// Communication
	fbReadWriteReq(sNetID := sNetID, nPort := nPort, nIdxGroup := nIdxGroup, tTimeOut := tTimeOut, aData := aStatIOLRecords);
	bStatTriggerExecute := bExecute AND NOT bStatTriggerExecuteMem;
	bStatTriggerExecuteMem := bExecute;
	bStatTriggerError := fbReadWriteReq.bError AND NOT bStatTriggerErrorMem;
	bStatTriggerErrorMem := fbReadWriteReq.bError;
// Timer
	fbInstTimeOut(IN:= bStatBusyMem, PT := tTimeOut);
// Error management
	IF stStatLastErrorCode.nBlockError <> cDEFAULT OR stStatLastErrorCode.nAdsReadError <> cDEFAULT OR stStatLastErrorCode.nAdsWriteError <> cDEFAULT THEN
		bDone := FALSE;
		bBusy := FALSE;
		bStatBusyMem := FALSE;
		bError := TRUE;
		stErrorCode := stStatLastErrorCode;
		stStatLastErrorCode.nBlockError := cDEFAULT;
		stStatLastErrorCode.nAdsReadError := cDEFAULT;
		stStatLastErrorCode.nAdsWriteError := cDEFAULT;
		stStatLastErrorCode.nIndex := 0;
		stStatLastErrorCode.nSubIndex := 0;
		nStatState := cSTATE_READY;
		RETURN;
	END_IF;
	IF bStatTriggerError THEN
		stStatLastErrorCode := fbReadWriteReq.stErrorCode;          // Error: ADS error
		RETURN;
	END_IF
	IF fbInstTimeOut.Q THEN
		stStatLastErrorCode.nIndex := fbReadWriteReq.stErrorCode.nIndex;
		stStatLastErrorCode.nSubIndex := fbReadWriteReq.stErrorCode.nSubIndex;
		stStatLastErrorCode.nBlockError := cERR_TIME_OUT;			// Error: Time out detected  
		RETURN;
	END_IF;
// Start R/W request
	IF bStatTriggerExecute AND NOT bStatBusyMem THEN
		bStatSource := FALSE; 
		nStatBitLength := 0; 
		nStatIndex := 0; 
		bDone := FALSE; 
		bBusy := TRUE; 
		bStatBusyMem := TRUE; 
		bError := FALSE; 
		stErrorCode.nBlockError := cDEFAULT; 
		stErrorCode.nAdsReadError := cDEFAULT; 
		stErrorCode.nAdsWriteError := cDEFAULT; 
		stErrorCode.nIndex := 0; 
		stErrorCode.nSubIndex := 0; 
		stStatLastErrorCode.nBlockError := cDEFAULT; 
		stStatLastErrorCode.nAdsReadError := cDEFAULT; 
		stStatLastErrorCode.nAdsWriteError := cDEFAULT; 
		stStatLastErrorCode.nIndex := 0; 
		stStatLastErrorCode.nSubIndex := 0; 
		bStatRWSave := bRW;
		nStatCommandIndex := 0;
		// Store input selection flags internally 
		aStatInputSelections[0] := stDeviceData.stSelection.stCommands.bCmdRestoreFactorySettings;
		aStatInputSelections[1] := stDeviceData.stSelection.stCommands.bCmdTeachApply;
		aStatInputSelections[2] := stDeviceData.stSelection.stCommands.bCmdSetpoint1SingleValueTeach;
		aStatInputSelections[3] := stDeviceData.stSelection.stCommands.bCmdSetpoint2SingleValueTeach;
		aStatInputSelections[4] := stDeviceData.stSelection.stCommands.bCmdTwoValueTeachTp1Sp1;
		aStatInputSelections[5] := stDeviceData.stSelection.stCommands.bCmdTwoValueTeachTp2Sp1;
		aStatInputSelections[6] := stDeviceData.stSelection.stCommands.bCmdTwoValueTeachTp1Sp2;
		aStatInputSelections[7] := stDeviceData.stSelection.stCommands.bCmdTwoValueTeachTp2Sp2;
		aStatInputSelections[8] := stDeviceData.stSelection.stCommands.bCmdSetpoint1DynamicTeachStart;
		aStatInputSelections[9] := stDeviceData.stSelection.stCommands.bCmdSetpoint1DynamicTeachStop;
		aStatInputSelections[10] := stDeviceData.stSelection.stCommands.bCmdSetpoint2DynamicTeachStart;
		aStatInputSelections[11] := stDeviceData.stSelection.stCommands.bCmdSetpoint2DynamicTeachStop;
		aStatInputSelections[12] := stDeviceData.stSelection.stCommands.bCmdTeachCancel;
		aStatInputSelections[13] := stDeviceData.stSelection.stCommands.bCmdSetAnalogOutputLowerLimit;
		aStatInputSelections[14] := stDeviceData.stSelection.stCommands.bCmdSetAnalogOutputUpperLimit;
		aStatInputSelections[15] := stDeviceData.stSelection.stCommands.bCmdResetDiagnosisInformation;
		aStatInputSelections[16] := stDeviceData.stSelection.stCommands.bCmdStopMeasurement;
		aStatInputSelections[17] := stDeviceData.stSelection.stCommands.bCmdStartMeasurement;
		aStatInputSelections[18] := stDeviceData.stSelection.stCommands.bCmdSingleMeasurement;
		aStatInputSelections[19] := stDeviceData.stSelection.stCommands.bCmdIoLink11SystemTestCommand240Event8DfeAppears;
		aStatInputSelections[20] := stDeviceData.stSelection.stCommands.bCmdIoLink11SystemTestCommand241Event8DfeDisappears;
		aStatInputSelections[21] := stDeviceData.stSelection.stCommands.bCmdIoLink11SystemTestCommand242Event8DffAppears;
		aStatInputSelections[22] := stDeviceData.stSelection.stCommands.bCmdIoLink11SystemTestCommand243Event8DffDisappears;
		aStatInputSelections[23] := stDeviceData.stSelection.stDirectParametersPage1.bAll;
		aStatInputSelections[24] := stDeviceData.stSelection.stDirectParametersPage1.bReserved_1;
		aStatInputSelections[25] := stDeviceData.stSelection.stDirectParametersPage1.bMasterCycleTime;
		aStatInputSelections[26] := stDeviceData.stSelection.stDirectParametersPage1.bMinCycleTime;
		aStatInputSelections[27] := stDeviceData.stSelection.stDirectParametersPage1.bMSequenceCapability;
		aStatInputSelections[28] := stDeviceData.stSelection.stDirectParametersPage1.bIoLinkRevisionId;
		aStatInputSelections[29] := stDeviceData.stSelection.stDirectParametersPage1.bProcessDataInputLength;
		aStatInputSelections[30] := stDeviceData.stSelection.stDirectParametersPage1.bProcessDataOutputLength;
		aStatInputSelections[31] := stDeviceData.stSelection.stDirectParametersPage1.bVendorId1;
		aStatInputSelections[32] := stDeviceData.stSelection.stDirectParametersPage1.bVendorId2;
		aStatInputSelections[33] := stDeviceData.stSelection.stDirectParametersPage1.bDeviceId1;
		aStatInputSelections[34] := stDeviceData.stSelection.stDirectParametersPage1.bDeviceId2;
		aStatInputSelections[35] := stDeviceData.stSelection.stDirectParametersPage1.bDeviceId3;
		aStatInputSelections[36] := stDeviceData.stSelection.stDirectParametersPage1.bReserved_13;
		aStatInputSelections[37] := stDeviceData.stSelection.stDirectParametersPage1.bReserved_14;
		aStatInputSelections[38] := stDeviceData.stSelection.stDirectParametersPage1.bReserved_15;
		aStatInputSelections[39] := stDeviceData.stSelection.stDirectParametersPage1.bSystemCommand;
		aStatInputSelections[40] := stDeviceData.stSelection.stDirectParametersPage2.bAll;
		aStatInputSelections[41] := stDeviceData.stSelection.stDirectParametersPage2.bDeviceSpecificParameter1;
		aStatInputSelections[42] := stDeviceData.stSelection.stDirectParametersPage2.bDeviceSpecificParameter2;
		aStatInputSelections[43] := stDeviceData.stSelection.stDirectParametersPage2.bDeviceSpecificParameter3;
		aStatInputSelections[44] := stDeviceData.stSelection.stDirectParametersPage2.bDeviceSpecificParameter4;
		aStatInputSelections[45] := stDeviceData.stSelection.stDirectParametersPage2.bDeviceSpecificParameter5;
		aStatInputSelections[46] := stDeviceData.stSelection.stDirectParametersPage2.bDeviceSpecificParameter6;
		aStatInputSelections[47] := stDeviceData.stSelection.stDirectParametersPage2.bDeviceSpecificParameter7;
		aStatInputSelections[48] := stDeviceData.stSelection.stDirectParametersPage2.bDeviceSpecificParameter8;
		aStatInputSelections[49] := stDeviceData.stSelection.stDirectParametersPage2.bDeviceSpecificParameter9;
		aStatInputSelections[50] := stDeviceData.stSelection.stDirectParametersPage2.bDeviceSpecificParameter10;
		aStatInputSelections[51] := stDeviceData.stSelection.stDirectParametersPage2.bDeviceSpecificParameter11;
		aStatInputSelections[52] := stDeviceData.stSelection.stDirectParametersPage2.bDeviceSpecificParameter12;
		aStatInputSelections[53] := stDeviceData.stSelection.stDirectParametersPage2.bDeviceSpecificParameter13;
		aStatInputSelections[54] := stDeviceData.stSelection.stDirectParametersPage2.bDeviceSpecificParameter14;
		aStatInputSelections[55] := stDeviceData.stSelection.stDirectParametersPage2.bDeviceSpecificParameter15;
		aStatInputSelections[56] := stDeviceData.stSelection.stDirectParametersPage2.bDeviceSpecificParameter16;
		aStatInputSelections[57] := stDeviceData.stSelection.bSystemCommand;
		aStatInputSelections[58] := stDeviceData.stSelection.stDeviceAccessLocks.bAll;
		aStatInputSelections[59] := stDeviceData.stSelection.bVendorName;
		aStatInputSelections[60] := stDeviceData.stSelection.bVendorText;
		aStatInputSelections[61] := stDeviceData.stSelection.bProductName;
		aStatInputSelections[62] := stDeviceData.stSelection.bProductId;
		aStatInputSelections[63] := stDeviceData.stSelection.bProductText;
		aStatInputSelections[64] := stDeviceData.stSelection.bFirmwareRevision;
		aStatInputSelections[65] := stDeviceData.stSelection.bApplicationSpecificTag;
		aStatInputSelections[66] := stDeviceData.stSelection.bErrorCount;
		aStatInputSelections[67] := stDeviceData.stSelection.bDeviceStatus;
		aStatInputSelections[68] := stDeviceData.stSelection.bTeachInSelect;
		aStatInputSelections[69] := stDeviceData.stSelection.stTeachState.bAll;
		aStatInputSelections[70] := stDeviceData.stSelection.stSetpoints_60.bAll;
		aStatInputSelections[71] := stDeviceData.stSelection.stSetpoints_60.bParam1Bdc1Q1;
		aStatInputSelections[72] := stDeviceData.stSelection.stSetpoints_60.bParam2Bdc1Q1;
		aStatInputSelections[73] := stDeviceData.stSelection.stSwitchpointBdc1.bAll;
		aStatInputSelections[74] := stDeviceData.stSelection.stSwitchpointBdc1.bLogic;
		aStatInputSelections[75] := stDeviceData.stSelection.stSwitchpointBdc1.bMode;
		aStatInputSelections[76] := stDeviceData.stSelection.stSwitchpointBdc1.bHysteresis;
		aStatInputSelections[77] := stDeviceData.stSelection.stSetpoints_62.bAll;
		aStatInputSelections[78] := stDeviceData.stSelection.stSetpoints_62.bParam1Bdc2Q2;
		aStatInputSelections[79] := stDeviceData.stSelection.stSetpoints_62.bParam2Bdc2Q2;
		aStatInputSelections[80] := stDeviceData.stSelection.stSwitchpointBdc2.bAll;
		aStatInputSelections[81] := stDeviceData.stSelection.stSwitchpointBdc2.bLogic;
		aStatInputSelections[82] := stDeviceData.stSelection.stSwitchpointBdc2.bMode;
		aStatInputSelections[83] := stDeviceData.stSelection.stSwitchpointBdc2.bHysteresis;
		aStatInputSelections[84] := stDeviceData.stSelection.bLot;
		aStatInputSelections[85] := stDeviceData.stSelection.bOnDelaySwitchingOutput;
		aStatInputSelections[86] := stDeviceData.stSelection.bOffDelaySwitchingOutput;
		aStatInputSelections[87] := stDeviceData.stSelection.bMultiIOPin4;
		aStatInputSelections[88] := stDeviceData.stSelection.bMultiIOPin2;
		aStatInputSelections[89] := stDeviceData.stSelection.stAnalogRange.bAll;
		aStatInputSelections[90] := stDeviceData.stSelection.stAnalogRange.bLowerLimit;
		aStatInputSelections[91] := stDeviceData.stSelection.stAnalogRange.bUpperLimit;
		aStatInputSelections[92] := stDeviceData.stSelection.bTemperatureCompensation;
		aStatInputSelections[93] := stDeviceData.stSelection.stTeachpointSp1_80.bAll;
		aStatInputSelections[94] := stDeviceData.stSelection.stTeachpointSp1_80.bTp1;
		aStatInputSelections[95] := stDeviceData.stSelection.stTeachpointSp1_80.bTp2;
		aStatInputSelections[96] := stDeviceData.stSelection.stTeachpointSp2_81.bAll;
		aStatInputSelections[97] := stDeviceData.stSelection.stTeachpointSp2_81.bTp1;
		aStatInputSelections[98] := stDeviceData.stSelection.stTeachpointSp2_81.bTp2;
		aStatInputSelections[99] := stDeviceData.stSelection.stTeachpointSp1_82.bAll;
		aStatInputSelections[100] := stDeviceData.stSelection.stTeachpointSp1_82.bTp1;
		aStatInputSelections[101] := stDeviceData.stSelection.stTeachpointSp1_82.bTp2;
		aStatInputSelections[102] := stDeviceData.stSelection.stTeachpointSp2_83.bAll;
		aStatInputSelections[103] := stDeviceData.stSelection.stTeachpointSp2_83.bTp1;
		aStatInputSelections[104] := stDeviceData.stSelection.stTeachpointSp2_83.bTp2;
		aStatInputSelections[105] := stDeviceData.stSelection.stProcessDataLimits.bAll;
		aStatInputSelections[106] := stDeviceData.stSelection.stProcessDataLimits.bLower;
		aStatInputSelections[107] := stDeviceData.stSelection.stProcessDataLimits.bUpper;
		aStatInputSelections[108] := stDeviceData.stSelection.bSwitchCounter;
		aStatInputSelections[109] := stDeviceData.stSelection.bTemperatureInternal;
		aStatInputSelections[110] := stDeviceData.stSelection.stNetwork.bAll;
		aStatInputSelections[111] := stDeviceData.stSelection.stNetwork.bRoleInNetwork;
		aStatInputSelections[112] := stDeviceData.stSelection.stNetwork.bDeviceNoMasterHighestNo;
		nStatState := cSTATE_INIT;
		RETURN; // Show the Busy-Flag for at least one PLC cycle 
	END_IF;
// Create command queue
	IF nStatState = cSTATE_INIT THEN
		// Check number of selected input selection bits
		nStatNumSelection := 0;
		FOR nTempLoopIndex := 0 TO cNUMBER_INPUTS DO
			IF aStatInputSelections[nTempLoopIndex] THEN
				nStatNumSelection := nStatNumSelection + 1;
			END_IF;
		END_FOR;
		IF nStatNumSelection = 0 THEN
			stStatLastErrorCode.nBlockError := cERR_EMPTY_SELECTION;
			RETURN;
		END_IF;
		// Create command queue
		FOR nTempLoopIndex := 0 TO cNUMBER_INPUTS DO
			aStatCommandQueue[nTempLoopIndex].nIndex := cEMPTY_COMMAND_QUEUE;
		END_FOR;
		nTempLoopIndex := 0;
		// stCommands - bCmdRestoreFactorySettings [BOOL] [WRITE_ONLY]
		IF aStatInputSelections[0] THEN
			aStatCommandQueue[nTempLoopIndex].nIndex := 32767;
			aStatCommandQueue[nTempLoopIndex].nSubIndex := 1;
			aStatCommandQueue[nTempLoopIndex].nBitLength := 8;
			nTempLoopIndex := nTempLoopIndex + 1;
		END_IF;
		// stCommands - bCmdTeachApply [BOOL] [WRITE_ONLY]
		IF aStatInputSelections[1] THEN
			aStatCommandQueue[nTempLoopIndex].nIndex := 32767;
			aStatCommandQueue[nTempLoopIndex].nSubIndex := 2;
			aStatCommandQueue[nTempLoopIndex].nBitLength := 8;
			nTempLoopIndex := nTempLoopIndex + 1;
		END_IF;
		// stCommands - bCmdSetpoint1SingleValueTeach [BOOL] [WRITE_ONLY]
		IF aStatInputSelections[2] THEN
			aStatCommandQueue[nTempLoopIndex].nIndex := 32767;
			aStatCommandQueue[nTempLoopIndex].nSubIndex := 3;
			aStatCommandQueue[nTempLoopIndex].nBitLength := 8;
			nTempLoopIndex := nTempLoopIndex + 1;
		END_IF;
		// stCommands - bCmdSetpoint2SingleValueTeach [BOOL] [WRITE_ONLY]
		IF aStatInputSelections[3] THEN
			aStatCommandQueue[nTempLoopIndex].nIndex := 32767;
			aStatCommandQueue[nTempLoopIndex].nSubIndex := 4;
			aStatCommandQueue[nTempLoopIndex].nBitLength := 8;
			nTempLoopIndex := nTempLoopIndex + 1;
		END_IF;
		// stCommands - bCmdTwoValueTeachTp1Sp1 [BOOL] [WRITE_ONLY]
		IF aStatInputSelections[4] THEN
			aStatCommandQueue[nTempLoopIndex].nIndex := 32767;
			aStatCommandQueue[nTempLoopIndex].nSubIndex := 5;
			aStatCommandQueue[nTempLoopIndex].nBitLength := 8;
			nTempLoopIndex := nTempLoopIndex + 1;
		END_IF;
		// stCommands - bCmdTwoValueTeachTp2Sp1 [BOOL] [WRITE_ONLY]
		IF aStatInputSelections[5] THEN
			aStatCommandQueue[nTempLoopIndex].nIndex := 32767;
			aStatCommandQueue[nTempLoopIndex].nSubIndex := 6;
			aStatCommandQueue[nTempLoopIndex].nBitLength := 8;
			nTempLoopIndex := nTempLoopIndex + 1;
		END_IF;
		// stCommands - bCmdTwoValueTeachTp1Sp2 [BOOL] [WRITE_ONLY]
		IF aStatInputSelections[6] THEN
			aStatCommandQueue[nTempLoopIndex].nIndex := 32767;
			aStatCommandQueue[nTempLoopIndex].nSubIndex := 7;
			aStatCommandQueue[nTempLoopIndex].nBitLength := 8;
			nTempLoopIndex := nTempLoopIndex + 1;
		END_IF;
		// stCommands - bCmdTwoValueTeachTp2Sp2 [BOOL] [WRITE_ONLY]
		IF aStatInputSelections[7] THEN
			aStatCommandQueue[nTempLoopIndex].nIndex := 32767;
			aStatCommandQueue[nTempLoopIndex].nSubIndex := 8;
			aStatCommandQueue[nTempLoopIndex].nBitLength := 8;
			nTempLoopIndex := nTempLoopIndex + 1;
		END_IF;
		// stCommands - bCmdSetpoint1DynamicTeachStart [BOOL] [WRITE_ONLY]
		IF aStatInputSelections[8] THEN
			aStatCommandQueue[nTempLoopIndex].nIndex := 32767;
			aStatCommandQueue[nTempLoopIndex].nSubIndex := 9;
			aStatCommandQueue[nTempLoopIndex].nBitLength := 8;
			nTempLoopIndex := nTempLoopIndex + 1;
		END_IF;
		// stCommands - bCmdSetpoint1DynamicTeachStop [BOOL] [WRITE_ONLY]
		IF aStatInputSelections[9] THEN
			aStatCommandQueue[nTempLoopIndex].nIndex := 32767;
			aStatCommandQueue[nTempLoopIndex].nSubIndex := 10;
			aStatCommandQueue[nTempLoopIndex].nBitLength := 8;
			nTempLoopIndex := nTempLoopIndex + 1;
		END_IF;
		// stCommands - bCmdSetpoint2DynamicTeachStart [BOOL] [WRITE_ONLY]
		IF aStatInputSelections[10] THEN
			aStatCommandQueue[nTempLoopIndex].nIndex := 32767;
			aStatCommandQueue[nTempLoopIndex].nSubIndex := 11;
			aStatCommandQueue[nTempLoopIndex].nBitLength := 8;
			nTempLoopIndex := nTempLoopIndex + 1;
		END_IF;
		// stCommands - bCmdSetpoint2DynamicTeachStop [BOOL] [WRITE_ONLY]
		IF aStatInputSelections[11] THEN
			aStatCommandQueue[nTempLoopIndex].nIndex := 32767;
			aStatCommandQueue[nTempLoopIndex].nSubIndex := 12;
			aStatCommandQueue[nTempLoopIndex].nBitLength := 8;
			nTempLoopIndex := nTempLoopIndex + 1;
		END_IF;
		// stCommands - bCmdTeachCancel [BOOL] [WRITE_ONLY]
		IF aStatInputSelections[12] THEN
			aStatCommandQueue[nTempLoopIndex].nIndex := 32767;
			aStatCommandQueue[nTempLoopIndex].nSubIndex := 13;
			aStatCommandQueue[nTempLoopIndex].nBitLength := 8;
			nTempLoopIndex := nTempLoopIndex + 1;
		END_IF;
		// stCommands - bCmdSetAnalogOutputLowerLimit [BOOL] [WRITE_ONLY]
		IF aStatInputSelections[13] THEN
			aStatCommandQueue[nTempLoopIndex].nIndex := 32767;
			aStatCommandQueue[nTempLoopIndex].nSubIndex := 14;
			aStatCommandQueue[nTempLoopIndex].nBitLength := 8;
			nTempLoopIndex := nTempLoopIndex + 1;
		END_IF;
		// stCommands - bCmdSetAnalogOutputUpperLimit [BOOL] [WRITE_ONLY]
		IF aStatInputSelections[14] THEN
			aStatCommandQueue[nTempLoopIndex].nIndex := 32767;
			aStatCommandQueue[nTempLoopIndex].nSubIndex := 15;
			aStatCommandQueue[nTempLoopIndex].nBitLength := 8;
			nTempLoopIndex := nTempLoopIndex + 1;
		END_IF;
		// stCommands - bCmdResetDiagnosisInformation [BOOL] [WRITE_ONLY]
		IF aStatInputSelections[15] THEN
			aStatCommandQueue[nTempLoopIndex].nIndex := 32767;
			aStatCommandQueue[nTempLoopIndex].nSubIndex := 16;
			aStatCommandQueue[nTempLoopIndex].nBitLength := 8;
			nTempLoopIndex := nTempLoopIndex + 1;
		END_IF;
		// stCommands - bCmdStopMeasurement [BOOL] [WRITE_ONLY]
		IF aStatInputSelections[16] THEN
			aStatCommandQueue[nTempLoopIndex].nIndex := 32767;
			aStatCommandQueue[nTempLoopIndex].nSubIndex := 17;
			aStatCommandQueue[nTempLoopIndex].nBitLength := 8;
			nTempLoopIndex := nTempLoopIndex + 1;
		END_IF;
		// stCommands - bCmdStartMeasurement [BOOL] [WRITE_ONLY]
		IF aStatInputSelections[17] THEN
			aStatCommandQueue[nTempLoopIndex].nIndex := 32767;
			aStatCommandQueue[nTempLoopIndex].nSubIndex := 18;
			aStatCommandQueue[nTempLoopIndex].nBitLength := 8;
			nTempLoopIndex := nTempLoopIndex + 1;
		END_IF;
		// stCommands - bCmdSingleMeasurement [BOOL] [WRITE_ONLY]
		IF aStatInputSelections[18] THEN
			aStatCommandQueue[nTempLoopIndex].nIndex := 32767;
			aStatCommandQueue[nTempLoopIndex].nSubIndex := 19;
			aStatCommandQueue[nTempLoopIndex].nBitLength := 8;
			nTempLoopIndex := nTempLoopIndex + 1;
		END_IF;
		// stCommands - bCmdIoLink11SystemTestCommand240Event8DfeAppears [BOOL] [WRITE_ONLY]
		IF aStatInputSelections[19] THEN
			aStatCommandQueue[nTempLoopIndex].nIndex := 32767;
			aStatCommandQueue[nTempLoopIndex].nSubIndex := 20;
			aStatCommandQueue[nTempLoopIndex].nBitLength := 8;
			nTempLoopIndex := nTempLoopIndex + 1;
		END_IF;
		// stCommands - bCmdIoLink11SystemTestCommand241Event8DfeDisappears [BOOL] [WRITE_ONLY]
		IF aStatInputSelections[20] THEN
			aStatCommandQueue[nTempLoopIndex].nIndex := 32767;
			aStatCommandQueue[nTempLoopIndex].nSubIndex := 21;
			aStatCommandQueue[nTempLoopIndex].nBitLength := 8;
			nTempLoopIndex := nTempLoopIndex + 1;
		END_IF;
		// stCommands - bCmdIoLink11SystemTestCommand242Event8DffAppears [BOOL] [WRITE_ONLY]
		IF aStatInputSelections[21] THEN
			aStatCommandQueue[nTempLoopIndex].nIndex := 32767;
			aStatCommandQueue[nTempLoopIndex].nSubIndex := 22;
			aStatCommandQueue[nTempLoopIndex].nBitLength := 8;
			nTempLoopIndex := nTempLoopIndex + 1;
		END_IF;
		// stCommands - bCmdIoLink11SystemTestCommand243Event8DffDisappears [BOOL] [WRITE_ONLY]
		IF aStatInputSelections[22] THEN
			aStatCommandQueue[nTempLoopIndex].nIndex := 32767;
			aStatCommandQueue[nTempLoopIndex].nSubIndex := 23;
			aStatCommandQueue[nTempLoopIndex].nBitLength := 8;
			nTempLoopIndex := nTempLoopIndex + 1;
		END_IF;
		// stDirectParametersPage1 - bAll [BOOL] [READ_WRITE]
		IF aStatInputSelections[23] THEN
			aStatCommandQueue[nTempLoopIndex].nIndex := 0;
			aStatCommandQueue[nTempLoopIndex].nSubIndex := 0;
			aStatCommandQueue[nTempLoopIndex].nBitLength := 128;
			nTempLoopIndex := nTempLoopIndex + 1;
		END_IF;
		// stDirectParametersPage1 - bReserved_1 [BOOL] [READ_ONLY]
		IF aStatInputSelections[24] THEN
			aStatCommandQueue[nTempLoopIndex].nIndex := 0;
			aStatCommandQueue[nTempLoopIndex].nSubIndex := 1;
			aStatCommandQueue[nTempLoopIndex].nBitLength := 8;
			nTempLoopIndex := nTempLoopIndex + 1;
		END_IF;
		// stDirectParametersPage1 - bMasterCycleTime [BOOL] [READ_ONLY]
		IF aStatInputSelections[25] THEN
			aStatCommandQueue[nTempLoopIndex].nIndex := 0;
			aStatCommandQueue[nTempLoopIndex].nSubIndex := 2;
			aStatCommandQueue[nTempLoopIndex].nBitLength := 8;
			nTempLoopIndex := nTempLoopIndex + 1;
		END_IF;
		// stDirectParametersPage1 - bMinCycleTime [BOOL] [READ_ONLY]
		IF aStatInputSelections[26] THEN
			aStatCommandQueue[nTempLoopIndex].nIndex := 0;
			aStatCommandQueue[nTempLoopIndex].nSubIndex := 3;
			aStatCommandQueue[nTempLoopIndex].nBitLength := 8;
			nTempLoopIndex := nTempLoopIndex + 1;
		END_IF;
		// stDirectParametersPage1 - bMSequenceCapability [BOOL] [READ_ONLY]
		IF aStatInputSelections[27] THEN
			aStatCommandQueue[nTempLoopIndex].nIndex := 0;
			aStatCommandQueue[nTempLoopIndex].nSubIndex := 4;
			aStatCommandQueue[nTempLoopIndex].nBitLength := 8;
			nTempLoopIndex := nTempLoopIndex + 1;
		END_IF;
		// stDirectParametersPage1 - bIoLinkRevisionId [BOOL] [READ_ONLY]
		IF aStatInputSelections[28] THEN
			aStatCommandQueue[nTempLoopIndex].nIndex := 0;
			aStatCommandQueue[nTempLoopIndex].nSubIndex := 5;
			aStatCommandQueue[nTempLoopIndex].nBitLength := 8;
			nTempLoopIndex := nTempLoopIndex + 1;
		END_IF;
		// stDirectParametersPage1 - bProcessDataInputLength [BOOL] [READ_ONLY]
		IF aStatInputSelections[29] THEN
			aStatCommandQueue[nTempLoopIndex].nIndex := 0;
			aStatCommandQueue[nTempLoopIndex].nSubIndex := 6;
			aStatCommandQueue[nTempLoopIndex].nBitLength := 8;
			nTempLoopIndex := nTempLoopIndex + 1;
		END_IF;
		// stDirectParametersPage1 - bProcessDataOutputLength [BOOL] [READ_ONLY]
		IF aStatInputSelections[30] THEN
			aStatCommandQueue[nTempLoopIndex].nIndex := 0;
			aStatCommandQueue[nTempLoopIndex].nSubIndex := 7;
			aStatCommandQueue[nTempLoopIndex].nBitLength := 8;
			nTempLoopIndex := nTempLoopIndex + 1;
		END_IF;
		// stDirectParametersPage1 - bVendorId1 [BOOL] [READ_ONLY]
		IF aStatInputSelections[31] THEN
			aStatCommandQueue[nTempLoopIndex].nIndex := 0;
			aStatCommandQueue[nTempLoopIndex].nSubIndex := 8;
			aStatCommandQueue[nTempLoopIndex].nBitLength := 8;
			nTempLoopIndex := nTempLoopIndex + 1;
		END_IF;
		// stDirectParametersPage1 - bVendorId2 [BOOL] [READ_ONLY]
		IF aStatInputSelections[32] THEN
			aStatCommandQueue[nTempLoopIndex].nIndex := 0;
			aStatCommandQueue[nTempLoopIndex].nSubIndex := 9;
			aStatCommandQueue[nTempLoopIndex].nBitLength := 8;
			nTempLoopIndex := nTempLoopIndex + 1;
		END_IF;
		// stDirectParametersPage1 - bDeviceId1 [BOOL] [READ_ONLY]
		IF aStatInputSelections[33] THEN
			aStatCommandQueue[nTempLoopIndex].nIndex := 0;
			aStatCommandQueue[nTempLoopIndex].nSubIndex := 10;
			aStatCommandQueue[nTempLoopIndex].nBitLength := 8;
			nTempLoopIndex := nTempLoopIndex + 1;
		END_IF;
		// stDirectParametersPage1 - bDeviceId2 [BOOL] [READ_ONLY]
		IF aStatInputSelections[34] THEN
			aStatCommandQueue[nTempLoopIndex].nIndex := 0;
			aStatCommandQueue[nTempLoopIndex].nSubIndex := 11;
			aStatCommandQueue[nTempLoopIndex].nBitLength := 8;
			nTempLoopIndex := nTempLoopIndex + 1;
		END_IF;
		// stDirectParametersPage1 - bDeviceId3 [BOOL] [READ_ONLY]
		IF aStatInputSelections[35] THEN
			aStatCommandQueue[nTempLoopIndex].nIndex := 0;
			aStatCommandQueue[nTempLoopIndex].nSubIndex := 12;
			aStatCommandQueue[nTempLoopIndex].nBitLength := 8;
			nTempLoopIndex := nTempLoopIndex + 1;
		END_IF;
		// stDirectParametersPage1 - bReserved_13 [BOOL] [READ_ONLY]
		IF aStatInputSelections[36] THEN
			aStatCommandQueue[nTempLoopIndex].nIndex := 0;
			aStatCommandQueue[nTempLoopIndex].nSubIndex := 13;
			aStatCommandQueue[nTempLoopIndex].nBitLength := 8;
			nTempLoopIndex := nTempLoopIndex + 1;
		END_IF;
		// stDirectParametersPage1 - bReserved_14 [BOOL] [READ_ONLY]
		IF aStatInputSelections[37] THEN
			aStatCommandQueue[nTempLoopIndex].nIndex := 0;
			aStatCommandQueue[nTempLoopIndex].nSubIndex := 14;
			aStatCommandQueue[nTempLoopIndex].nBitLength := 8;
			nTempLoopIndex := nTempLoopIndex + 1;
		END_IF;
		// stDirectParametersPage1 - bReserved_15 [BOOL] [READ_ONLY]
		IF aStatInputSelections[38] THEN
			aStatCommandQueue[nTempLoopIndex].nIndex := 0;
			aStatCommandQueue[nTempLoopIndex].nSubIndex := 15;
			aStatCommandQueue[nTempLoopIndex].nBitLength := 8;
			nTempLoopIndex := nTempLoopIndex + 1;
		END_IF;
		// stDirectParametersPage1 - bSystemCommand [BOOL] [WRITE_ONLY]
		IF aStatInputSelections[39] THEN
			aStatCommandQueue[nTempLoopIndex].nIndex := 0;
			aStatCommandQueue[nTempLoopIndex].nSubIndex := 16;
			aStatCommandQueue[nTempLoopIndex].nBitLength := 8;
			nTempLoopIndex := nTempLoopIndex + 1;
		END_IF;
		// stDirectParametersPage2 - bAll [BOOL] [READ_WRITE]
		IF aStatInputSelections[40] THEN
			aStatCommandQueue[nTempLoopIndex].nIndex := 1;
			aStatCommandQueue[nTempLoopIndex].nSubIndex := 0;
			aStatCommandQueue[nTempLoopIndex].nBitLength := 128;
			nTempLoopIndex := nTempLoopIndex + 1;
		END_IF;
		// stDirectParametersPage2 - bDeviceSpecificParameter1 [BOOL] [READ_WRITE]
		IF aStatInputSelections[41] THEN
			aStatCommandQueue[nTempLoopIndex].nIndex := 1;
			aStatCommandQueue[nTempLoopIndex].nSubIndex := 1;
			aStatCommandQueue[nTempLoopIndex].nBitLength := 8;
			nTempLoopIndex := nTempLoopIndex + 1;
		END_IF;
		// stDirectParametersPage2 - bDeviceSpecificParameter2 [BOOL] [READ_WRITE]
		IF aStatInputSelections[42] THEN
			aStatCommandQueue[nTempLoopIndex].nIndex := 1;
			aStatCommandQueue[nTempLoopIndex].nSubIndex := 2;
			aStatCommandQueue[nTempLoopIndex].nBitLength := 8;
			nTempLoopIndex := nTempLoopIndex + 1;
		END_IF;
		// stDirectParametersPage2 - bDeviceSpecificParameter3 [BOOL] [READ_WRITE]
		IF aStatInputSelections[43] THEN
			aStatCommandQueue[nTempLoopIndex].nIndex := 1;
			aStatCommandQueue[nTempLoopIndex].nSubIndex := 3;
			aStatCommandQueue[nTempLoopIndex].nBitLength := 8;
			nTempLoopIndex := nTempLoopIndex + 1;
		END_IF;
		// stDirectParametersPage2 - bDeviceSpecificParameter4 [BOOL] [READ_WRITE]
		IF aStatInputSelections[44] THEN
			aStatCommandQueue[nTempLoopIndex].nIndex := 1;
			aStatCommandQueue[nTempLoopIndex].nSubIndex := 4;
			aStatCommandQueue[nTempLoopIndex].nBitLength := 8;
			nTempLoopIndex := nTempLoopIndex + 1;
		END_IF;
		// stDirectParametersPage2 - bDeviceSpecificParameter5 [BOOL] [READ_WRITE]
		IF aStatInputSelections[45] THEN
			aStatCommandQueue[nTempLoopIndex].nIndex := 1;
			aStatCommandQueue[nTempLoopIndex].nSubIndex := 5;
			aStatCommandQueue[nTempLoopIndex].nBitLength := 8;
			nTempLoopIndex := nTempLoopIndex + 1;
		END_IF;
		// stDirectParametersPage2 - bDeviceSpecificParameter6 [BOOL] [READ_WRITE]
		IF aStatInputSelections[46] THEN
			aStatCommandQueue[nTempLoopIndex].nIndex := 1;
			aStatCommandQueue[nTempLoopIndex].nSubIndex := 6;
			aStatCommandQueue[nTempLoopIndex].nBitLength := 8;
			nTempLoopIndex := nTempLoopIndex + 1;
		END_IF;
		// stDirectParametersPage2 - bDeviceSpecificParameter7 [BOOL] [READ_WRITE]
		IF aStatInputSelections[47] THEN
			aStatCommandQueue[nTempLoopIndex].nIndex := 1;
			aStatCommandQueue[nTempLoopIndex].nSubIndex := 7;
			aStatCommandQueue[nTempLoopIndex].nBitLength := 8;
			nTempLoopIndex := nTempLoopIndex + 1;
		END_IF;
		// stDirectParametersPage2 - bDeviceSpecificParameter8 [BOOL] [READ_WRITE]
		IF aStatInputSelections[48] THEN
			aStatCommandQueue[nTempLoopIndex].nIndex := 1;
			aStatCommandQueue[nTempLoopIndex].nSubIndex := 8;
			aStatCommandQueue[nTempLoopIndex].nBitLength := 8;
			nTempLoopIndex := nTempLoopIndex + 1;
		END_IF;
		// stDirectParametersPage2 - bDeviceSpecificParameter9 [BOOL] [READ_WRITE]
		IF aStatInputSelections[49] THEN
			aStatCommandQueue[nTempLoopIndex].nIndex := 1;
			aStatCommandQueue[nTempLoopIndex].nSubIndex := 9;
			aStatCommandQueue[nTempLoopIndex].nBitLength := 8;
			nTempLoopIndex := nTempLoopIndex + 1;
		END_IF;
		// stDirectParametersPage2 - bDeviceSpecificParameter10 [BOOL] [READ_WRITE]
		IF aStatInputSelections[50] THEN
			aStatCommandQueue[nTempLoopIndex].nIndex := 1;
			aStatCommandQueue[nTempLoopIndex].nSubIndex := 10;
			aStatCommandQueue[nTempLoopIndex].nBitLength := 8;
			nTempLoopIndex := nTempLoopIndex + 1;
		END_IF;
		// stDirectParametersPage2 - bDeviceSpecificParameter11 [BOOL] [READ_WRITE]
		IF aStatInputSelections[51] THEN
			aStatCommandQueue[nTempLoopIndex].nIndex := 1;
			aStatCommandQueue[nTempLoopIndex].nSubIndex := 11;
			aStatCommandQueue[nTempLoopIndex].nBitLength := 8;
			nTempLoopIndex := nTempLoopIndex + 1;
		END_IF;
		// stDirectParametersPage2 - bDeviceSpecificParameter12 [BOOL] [READ_WRITE]
		IF aStatInputSelections[52] THEN
			aStatCommandQueue[nTempLoopIndex].nIndex := 1;
			aStatCommandQueue[nTempLoopIndex].nSubIndex := 12;
			aStatCommandQueue[nTempLoopIndex].nBitLength := 8;
			nTempLoopIndex := nTempLoopIndex + 1;
		END_IF;
		// stDirectParametersPage2 - bDeviceSpecificParameter13 [BOOL] [READ_WRITE]
		IF aStatInputSelections[53] THEN
			aStatCommandQueue[nTempLoopIndex].nIndex := 1;
			aStatCommandQueue[nTempLoopIndex].nSubIndex := 13;
			aStatCommandQueue[nTempLoopIndex].nBitLength := 8;
			nTempLoopIndex := nTempLoopIndex + 1;
		END_IF;
		// stDirectParametersPage2 - bDeviceSpecificParameter14 [BOOL] [READ_WRITE]
		IF aStatInputSelections[54] THEN
			aStatCommandQueue[nTempLoopIndex].nIndex := 1;
			aStatCommandQueue[nTempLoopIndex].nSubIndex := 14;
			aStatCommandQueue[nTempLoopIndex].nBitLength := 8;
			nTempLoopIndex := nTempLoopIndex + 1;
		END_IF;
		// stDirectParametersPage2 - bDeviceSpecificParameter15 [BOOL] [READ_WRITE]
		IF aStatInputSelections[55] THEN
			aStatCommandQueue[nTempLoopIndex].nIndex := 1;
			aStatCommandQueue[nTempLoopIndex].nSubIndex := 15;
			aStatCommandQueue[nTempLoopIndex].nBitLength := 8;
			nTempLoopIndex := nTempLoopIndex + 1;
		END_IF;
		// stDirectParametersPage2 - bDeviceSpecificParameter16 [BOOL] [READ_WRITE]
		IF aStatInputSelections[56] THEN
			aStatCommandQueue[nTempLoopIndex].nIndex := 1;
			aStatCommandQueue[nTempLoopIndex].nSubIndex := 16;
			aStatCommandQueue[nTempLoopIndex].nBitLength := 8;
			nTempLoopIndex := nTempLoopIndex + 1;
		END_IF;
		// bSystemCommand [BOOL] [WRITE_ONLY]
		IF aStatInputSelections[57] THEN
			aStatCommandQueue[nTempLoopIndex].nIndex := 2;
			aStatCommandQueue[nTempLoopIndex].nSubIndex := 0;
			aStatCommandQueue[nTempLoopIndex].nBitLength := 8;
			nTempLoopIndex := nTempLoopIndex + 1;
		END_IF;
		// stDeviceAccessLocks - bAll [BOOL] [READ_WRITE]
		IF aStatInputSelections[58] THEN
			aStatCommandQueue[nTempLoopIndex].nIndex := 12;
			aStatCommandQueue[nTempLoopIndex].nSubIndex := 0;
			aStatCommandQueue[nTempLoopIndex].nBitLength := 16;
			nTempLoopIndex := nTempLoopIndex + 1;
		END_IF;
		// bVendorName [BOOL] [READ_ONLY]
		IF aStatInputSelections[59] THEN
			aStatCommandQueue[nTempLoopIndex].nIndex := 16;
			aStatCommandQueue[nTempLoopIndex].nSubIndex := 0;
			aStatCommandQueue[nTempLoopIndex].nBitLength := 512;
			nTempLoopIndex := nTempLoopIndex + 1;
		END_IF;
		// bVendorText [BOOL] [READ_ONLY]
		IF aStatInputSelections[60] THEN
			aStatCommandQueue[nTempLoopIndex].nIndex := 17;
			aStatCommandQueue[nTempLoopIndex].nSubIndex := 0;
			aStatCommandQueue[nTempLoopIndex].nBitLength := 512;
			nTempLoopIndex := nTempLoopIndex + 1;
		END_IF;
		// bProductName [BOOL] [READ_ONLY]
		IF aStatInputSelections[61] THEN
			aStatCommandQueue[nTempLoopIndex].nIndex := 18;
			aStatCommandQueue[nTempLoopIndex].nSubIndex := 0;
			aStatCommandQueue[nTempLoopIndex].nBitLength := 512;
			nTempLoopIndex := nTempLoopIndex + 1;
		END_IF;
		// bProductId [BOOL] [READ_ONLY]
		IF aStatInputSelections[62] THEN
			aStatCommandQueue[nTempLoopIndex].nIndex := 19;
			aStatCommandQueue[nTempLoopIndex].nSubIndex := 0;
			aStatCommandQueue[nTempLoopIndex].nBitLength := 512;
			nTempLoopIndex := nTempLoopIndex + 1;
		END_IF;
		// bProductText [BOOL] [READ_ONLY]
		IF aStatInputSelections[63] THEN
			aStatCommandQueue[nTempLoopIndex].nIndex := 20;
			aStatCommandQueue[nTempLoopIndex].nSubIndex := 0;
			aStatCommandQueue[nTempLoopIndex].nBitLength := 512;
			nTempLoopIndex := nTempLoopIndex + 1;
		END_IF;
		// bFirmwareRevision [BOOL] [READ_ONLY]
		IF aStatInputSelections[64] THEN
			aStatCommandQueue[nTempLoopIndex].nIndex := 23;
			aStatCommandQueue[nTempLoopIndex].nSubIndex := 0;
			aStatCommandQueue[nTempLoopIndex].nBitLength := 512;
			nTempLoopIndex := nTempLoopIndex + 1;
		END_IF;
		// bApplicationSpecificTag [BOOL] [READ_WRITE]
		IF aStatInputSelections[65] THEN
			aStatCommandQueue[nTempLoopIndex].nIndex := 24;
			aStatCommandQueue[nTempLoopIndex].nSubIndex := 0;
			aStatCommandQueue[nTempLoopIndex].nBitLength := 256;
			nTempLoopIndex := nTempLoopIndex + 1;
		END_IF;
		// bErrorCount [BOOL] [READ_ONLY]
		IF aStatInputSelections[66] THEN
			aStatCommandQueue[nTempLoopIndex].nIndex := 32;
			aStatCommandQueue[nTempLoopIndex].nSubIndex := 0;
			aStatCommandQueue[nTempLoopIndex].nBitLength := 16;
			nTempLoopIndex := nTempLoopIndex + 1;
		END_IF;
		// bDeviceStatus [BOOL] [READ_ONLY]
		IF aStatInputSelections[67] THEN
			aStatCommandQueue[nTempLoopIndex].nIndex := 36;
			aStatCommandQueue[nTempLoopIndex].nSubIndex := 0;
			aStatCommandQueue[nTempLoopIndex].nBitLength := 8;
			nTempLoopIndex := nTempLoopIndex + 1;
		END_IF;
		// bTeachInSelect [BOOL] [READ_WRITE]
		IF aStatInputSelections[68] THEN
			aStatCommandQueue[nTempLoopIndex].nIndex := 58;
			aStatCommandQueue[nTempLoopIndex].nSubIndex := 0;
			aStatCommandQueue[nTempLoopIndex].nBitLength := 8;
			nTempLoopIndex := nTempLoopIndex + 1;
		END_IF;
		// stTeachState - bAll [BOOL] [READ_ONLY]
		IF aStatInputSelections[69] THEN
			aStatCommandQueue[nTempLoopIndex].nIndex := 59;
			aStatCommandQueue[nTempLoopIndex].nSubIndex := 0;
			aStatCommandQueue[nTempLoopIndex].nBitLength := 8;
			nTempLoopIndex := nTempLoopIndex + 1;
		END_IF;
		// stSetpoints_60 - bAll [BOOL] [READ_WRITE]
		IF aStatInputSelections[70] THEN
			aStatCommandQueue[nTempLoopIndex].nIndex := 60;
			aStatCommandQueue[nTempLoopIndex].nSubIndex := 0;
			aStatCommandQueue[nTempLoopIndex].nBitLength := 32;
			nTempLoopIndex := nTempLoopIndex + 1;
		END_IF;
		// stSetpoints_60 - bParam1Bdc1Q1 [BOOL] [READ_WRITE]
		IF aStatInputSelections[71] THEN
			aStatCommandQueue[nTempLoopIndex].nIndex := 60;
			aStatCommandQueue[nTempLoopIndex].nSubIndex := 1;
			aStatCommandQueue[nTempLoopIndex].nBitLength := 16;
			nTempLoopIndex := nTempLoopIndex + 1;
		END_IF;
		// stSetpoints_60 - bParam2Bdc1Q1 [BOOL] [READ_WRITE]
		IF aStatInputSelections[72] THEN
			aStatCommandQueue[nTempLoopIndex].nIndex := 60;
			aStatCommandQueue[nTempLoopIndex].nSubIndex := 2;
			aStatCommandQueue[nTempLoopIndex].nBitLength := 16;
			nTempLoopIndex := nTempLoopIndex + 1;
		END_IF;
		// stSwitchpointBdc1 - bAll [BOOL] [READ_WRITE]
		IF aStatInputSelections[73] THEN
			aStatCommandQueue[nTempLoopIndex].nIndex := 61;
			aStatCommandQueue[nTempLoopIndex].nSubIndex := 0;
			aStatCommandQueue[nTempLoopIndex].nBitLength := 32;
			nTempLoopIndex := nTempLoopIndex + 1;
		END_IF;
		// stSwitchpointBdc1 - bLogic [BOOL] [READ_WRITE]
		IF aStatInputSelections[74] THEN
			aStatCommandQueue[nTempLoopIndex].nIndex := 61;
			aStatCommandQueue[nTempLoopIndex].nSubIndex := 1;
			aStatCommandQueue[nTempLoopIndex].nBitLength := 8;
			nTempLoopIndex := nTempLoopIndex + 1;
		END_IF;
		// stSwitchpointBdc1 - bMode [BOOL] [READ_WRITE]
		IF aStatInputSelections[75] THEN
			aStatCommandQueue[nTempLoopIndex].nIndex := 61;
			aStatCommandQueue[nTempLoopIndex].nSubIndex := 2;
			aStatCommandQueue[nTempLoopIndex].nBitLength := 8;
			nTempLoopIndex := nTempLoopIndex + 1;
		END_IF;
		// stSwitchpointBdc1 - bHysteresis [BOOL] [READ_WRITE]
		IF aStatInputSelections[76] THEN
			aStatCommandQueue[nTempLoopIndex].nIndex := 61;
			aStatCommandQueue[nTempLoopIndex].nSubIndex := 3;
			aStatCommandQueue[nTempLoopIndex].nBitLength := 16;
			nTempLoopIndex := nTempLoopIndex + 1;
		END_IF;
		// stSetpoints_62 - bAll [BOOL] [READ_WRITE]
		IF aStatInputSelections[77] THEN
			aStatCommandQueue[nTempLoopIndex].nIndex := 62;
			aStatCommandQueue[nTempLoopIndex].nSubIndex := 0;
			aStatCommandQueue[nTempLoopIndex].nBitLength := 32;
			nTempLoopIndex := nTempLoopIndex + 1;
		END_IF;
		// stSetpoints_62 - bParam1Bdc2Q2 [BOOL] [READ_WRITE]
		IF aStatInputSelections[78] THEN
			aStatCommandQueue[nTempLoopIndex].nIndex := 62;
			aStatCommandQueue[nTempLoopIndex].nSubIndex := 1;
			aStatCommandQueue[nTempLoopIndex].nBitLength := 16;
			nTempLoopIndex := nTempLoopIndex + 1;
		END_IF;
		// stSetpoints_62 - bParam2Bdc2Q2 [BOOL] [READ_WRITE]
		IF aStatInputSelections[79] THEN
			aStatCommandQueue[nTempLoopIndex].nIndex := 62;
			aStatCommandQueue[nTempLoopIndex].nSubIndex := 2;
			aStatCommandQueue[nTempLoopIndex].nBitLength := 16;
			nTempLoopIndex := nTempLoopIndex + 1;
		END_IF;
		// stSwitchpointBdc2 - bAll [BOOL] [READ_WRITE]
		IF aStatInputSelections[80] THEN
			aStatCommandQueue[nTempLoopIndex].nIndex := 63;
			aStatCommandQueue[nTempLoopIndex].nSubIndex := 0;
			aStatCommandQueue[nTempLoopIndex].nBitLength := 32;
			nTempLoopIndex := nTempLoopIndex + 1;
		END_IF;
		// stSwitchpointBdc2 - bLogic [BOOL] [READ_WRITE]
		IF aStatInputSelections[81] THEN
			aStatCommandQueue[nTempLoopIndex].nIndex := 63;
			aStatCommandQueue[nTempLoopIndex].nSubIndex := 1;
			aStatCommandQueue[nTempLoopIndex].nBitLength := 8;
			nTempLoopIndex := nTempLoopIndex + 1;
		END_IF;
		// stSwitchpointBdc2 - bMode [BOOL] [READ_WRITE]
		IF aStatInputSelections[82] THEN
			aStatCommandQueue[nTempLoopIndex].nIndex := 63;
			aStatCommandQueue[nTempLoopIndex].nSubIndex := 2;
			aStatCommandQueue[nTempLoopIndex].nBitLength := 8;
			nTempLoopIndex := nTempLoopIndex + 1;
		END_IF;
		// stSwitchpointBdc2 - bHysteresis [BOOL] [READ_WRITE]
		IF aStatInputSelections[83] THEN
			aStatCommandQueue[nTempLoopIndex].nIndex := 63;
			aStatCommandQueue[nTempLoopIndex].nSubIndex := 3;
			aStatCommandQueue[nTempLoopIndex].nBitLength := 16;
			nTempLoopIndex := nTempLoopIndex + 1;
		END_IF;
		// bLot [BOOL] [READ_ONLY]
		IF aStatInputSelections[84] THEN
			aStatCommandQueue[nTempLoopIndex].nIndex := 64;
			aStatCommandQueue[nTempLoopIndex].nSubIndex := 0;
			aStatCommandQueue[nTempLoopIndex].nBitLength := 128;
			nTempLoopIndex := nTempLoopIndex + 1;
		END_IF;
		// bOnDelaySwitchingOutput [BOOL] [READ_WRITE]
		IF aStatInputSelections[85] THEN
			aStatCommandQueue[nTempLoopIndex].nIndex := 66;
			aStatCommandQueue[nTempLoopIndex].nSubIndex := 0;
			aStatCommandQueue[nTempLoopIndex].nBitLength := 16;
			nTempLoopIndex := nTempLoopIndex + 1;
		END_IF;
		// bOffDelaySwitchingOutput [BOOL] [READ_WRITE]
		IF aStatInputSelections[86] THEN
			aStatCommandQueue[nTempLoopIndex].nIndex := 67;
			aStatCommandQueue[nTempLoopIndex].nSubIndex := 0;
			aStatCommandQueue[nTempLoopIndex].nBitLength := 16;
			nTempLoopIndex := nTempLoopIndex + 1;
		END_IF;
		// bMultiIOPin4 [BOOL] [READ_WRITE]
		IF aStatInputSelections[87] THEN
			aStatCommandQueue[nTempLoopIndex].nIndex := 70;
			aStatCommandQueue[nTempLoopIndex].nSubIndex := 0;
			aStatCommandQueue[nTempLoopIndex].nBitLength := 8;
			nTempLoopIndex := nTempLoopIndex + 1;
		END_IF;
		// bMultiIOPin2 [BOOL] [READ_WRITE]
		IF aStatInputSelections[88] THEN
			aStatCommandQueue[nTempLoopIndex].nIndex := 71;
			aStatCommandQueue[nTempLoopIndex].nSubIndex := 0;
			aStatCommandQueue[nTempLoopIndex].nBitLength := 8;
			nTempLoopIndex := nTempLoopIndex + 1;
		END_IF;
		// stAnalogRange - bAll [BOOL] [READ_WRITE]
		IF aStatInputSelections[89] THEN
			aStatCommandQueue[nTempLoopIndex].nIndex := 72;
			aStatCommandQueue[nTempLoopIndex].nSubIndex := 0;
			aStatCommandQueue[nTempLoopIndex].nBitLength := 32;
			nTempLoopIndex := nTempLoopIndex + 1;
		END_IF;
		// stAnalogRange - bLowerLimit [BOOL] [READ_WRITE]
		IF aStatInputSelections[90] THEN
			aStatCommandQueue[nTempLoopIndex].nIndex := 72;
			aStatCommandQueue[nTempLoopIndex].nSubIndex := 1;
			aStatCommandQueue[nTempLoopIndex].nBitLength := 16;
			nTempLoopIndex := nTempLoopIndex + 1;
		END_IF;
		// stAnalogRange - bUpperLimit [BOOL] [READ_WRITE]
		IF aStatInputSelections[91] THEN
			aStatCommandQueue[nTempLoopIndex].nIndex := 72;
			aStatCommandQueue[nTempLoopIndex].nSubIndex := 2;
			aStatCommandQueue[nTempLoopIndex].nBitLength := 16;
			nTempLoopIndex := nTempLoopIndex + 1;
		END_IF;
		// bTemperatureCompensation [BOOL] [READ_WRITE]
		IF aStatInputSelections[92] THEN
			aStatCommandQueue[nTempLoopIndex].nIndex := 74;
			aStatCommandQueue[nTempLoopIndex].nSubIndex := 0;
			aStatCommandQueue[nTempLoopIndex].nBitLength := 8;
			nTempLoopIndex := nTempLoopIndex + 1;
		END_IF;
		// stTeachpointSp1_80 - bAll [BOOL] [READ_ONLY]
		IF aStatInputSelections[93] THEN
			aStatCommandQueue[nTempLoopIndex].nIndex := 80;
			aStatCommandQueue[nTempLoopIndex].nSubIndex := 0;
			aStatCommandQueue[nTempLoopIndex].nBitLength := 32;
			nTempLoopIndex := nTempLoopIndex + 1;
		END_IF;
		// stTeachpointSp1_80 - bTp1 [BOOL] [READ_ONLY]
		IF aStatInputSelections[94] THEN
			aStatCommandQueue[nTempLoopIndex].nIndex := 80;
			aStatCommandQueue[nTempLoopIndex].nSubIndex := 1;
			aStatCommandQueue[nTempLoopIndex].nBitLength := 16;
			nTempLoopIndex := nTempLoopIndex + 1;
		END_IF;
		// stTeachpointSp1_80 - bTp2 [BOOL] [READ_ONLY]
		IF aStatInputSelections[95] THEN
			aStatCommandQueue[nTempLoopIndex].nIndex := 80;
			aStatCommandQueue[nTempLoopIndex].nSubIndex := 2;
			aStatCommandQueue[nTempLoopIndex].nBitLength := 16;
			nTempLoopIndex := nTempLoopIndex + 1;
		END_IF;
		// stTeachpointSp2_81 - bAll [BOOL] [READ_ONLY]
		IF aStatInputSelections[96] THEN
			aStatCommandQueue[nTempLoopIndex].nIndex := 81;
			aStatCommandQueue[nTempLoopIndex].nSubIndex := 0;
			aStatCommandQueue[nTempLoopIndex].nBitLength := 32;
			nTempLoopIndex := nTempLoopIndex + 1;
		END_IF;
		// stTeachpointSp2_81 - bTp1 [BOOL] [READ_ONLY]
		IF aStatInputSelections[97] THEN
			aStatCommandQueue[nTempLoopIndex].nIndex := 81;
			aStatCommandQueue[nTempLoopIndex].nSubIndex := 1;
			aStatCommandQueue[nTempLoopIndex].nBitLength := 16;
			nTempLoopIndex := nTempLoopIndex + 1;
		END_IF;
		// stTeachpointSp2_81 - bTp2 [BOOL] [READ_ONLY]
		IF aStatInputSelections[98] THEN
			aStatCommandQueue[nTempLoopIndex].nIndex := 81;
			aStatCommandQueue[nTempLoopIndex].nSubIndex := 2;
			aStatCommandQueue[nTempLoopIndex].nBitLength := 16;
			nTempLoopIndex := nTempLoopIndex + 1;
		END_IF;
		// stTeachpointSp1_82 - bAll [BOOL] [READ_ONLY]
		IF aStatInputSelections[99] THEN
			aStatCommandQueue[nTempLoopIndex].nIndex := 82;
			aStatCommandQueue[nTempLoopIndex].nSubIndex := 0;
			aStatCommandQueue[nTempLoopIndex].nBitLength := 32;
			nTempLoopIndex := nTempLoopIndex + 1;
		END_IF;
		// stTeachpointSp1_82 - bTp1 [BOOL] [READ_ONLY]
		IF aStatInputSelections[100] THEN
			aStatCommandQueue[nTempLoopIndex].nIndex := 82;
			aStatCommandQueue[nTempLoopIndex].nSubIndex := 1;
			aStatCommandQueue[nTempLoopIndex].nBitLength := 16;
			nTempLoopIndex := nTempLoopIndex + 1;
		END_IF;
		// stTeachpointSp1_82 - bTp2 [BOOL] [READ_ONLY]
		IF aStatInputSelections[101] THEN
			aStatCommandQueue[nTempLoopIndex].nIndex := 82;
			aStatCommandQueue[nTempLoopIndex].nSubIndex := 2;
			aStatCommandQueue[nTempLoopIndex].nBitLength := 16;
			nTempLoopIndex := nTempLoopIndex + 1;
		END_IF;
		// stTeachpointSp2_83 - bAll [BOOL] [READ_ONLY]
		IF aStatInputSelections[102] THEN
			aStatCommandQueue[nTempLoopIndex].nIndex := 83;
			aStatCommandQueue[nTempLoopIndex].nSubIndex := 0;
			aStatCommandQueue[nTempLoopIndex].nBitLength := 32;
			nTempLoopIndex := nTempLoopIndex + 1;
		END_IF;
		// stTeachpointSp2_83 - bTp1 [BOOL] [READ_ONLY]
		IF aStatInputSelections[103] THEN
			aStatCommandQueue[nTempLoopIndex].nIndex := 83;
			aStatCommandQueue[nTempLoopIndex].nSubIndex := 1;
			aStatCommandQueue[nTempLoopIndex].nBitLength := 16;
			nTempLoopIndex := nTempLoopIndex + 1;
		END_IF;
		// stTeachpointSp2_83 - bTp2 [BOOL] [READ_ONLY]
		IF aStatInputSelections[104] THEN
			aStatCommandQueue[nTempLoopIndex].nIndex := 83;
			aStatCommandQueue[nTempLoopIndex].nSubIndex := 2;
			aStatCommandQueue[nTempLoopIndex].nBitLength := 16;
			nTempLoopIndex := nTempLoopIndex + 1;
		END_IF;
		// stProcessDataLimits - bAll [BOOL] [READ_ONLY]
		IF aStatInputSelections[105] THEN
			aStatCommandQueue[nTempLoopIndex].nIndex := 84;
			aStatCommandQueue[nTempLoopIndex].nSubIndex := 0;
			aStatCommandQueue[nTempLoopIndex].nBitLength := 32;
			nTempLoopIndex := nTempLoopIndex + 1;
		END_IF;
		// stProcessDataLimits - bLower [BOOL] [READ_ONLY]
		IF aStatInputSelections[106] THEN
			aStatCommandQueue[nTempLoopIndex].nIndex := 84;
			aStatCommandQueue[nTempLoopIndex].nSubIndex := 1;
			aStatCommandQueue[nTempLoopIndex].nBitLength := 16;
			nTempLoopIndex := nTempLoopIndex + 1;
		END_IF;
		// stProcessDataLimits - bUpper [BOOL] [READ_ONLY]
		IF aStatInputSelections[107] THEN
			aStatCommandQueue[nTempLoopIndex].nIndex := 84;
			aStatCommandQueue[nTempLoopIndex].nSubIndex := 2;
			aStatCommandQueue[nTempLoopIndex].nBitLength := 16;
			nTempLoopIndex := nTempLoopIndex + 1;
		END_IF;
		// bSwitchCounter [BOOL] [READ_ONLY]
		IF aStatInputSelections[108] THEN
			aStatCommandQueue[nTempLoopIndex].nIndex := 85;
			aStatCommandQueue[nTempLoopIndex].nSubIndex := 0;
			aStatCommandQueue[nTempLoopIndex].nBitLength := 32;
			nTempLoopIndex := nTempLoopIndex + 1;
		END_IF;
		// bTemperatureInternal [BOOL] [READ_ONLY]
		IF aStatInputSelections[109] THEN
			aStatCommandQueue[nTempLoopIndex].nIndex := 86;
			aStatCommandQueue[nTempLoopIndex].nSubIndex := 0;
			aStatCommandQueue[nTempLoopIndex].nBitLength := 16;
			nTempLoopIndex := nTempLoopIndex + 1;
		END_IF;
		// stNetwork - bAll [BOOL] [READ_WRITE]
		IF aStatInputSelections[110] THEN
			aStatCommandQueue[nTempLoopIndex].nIndex := 88;
			aStatCommandQueue[nTempLoopIndex].nSubIndex := 0;
			aStatCommandQueue[nTempLoopIndex].nBitLength := 16;
			nTempLoopIndex := nTempLoopIndex + 1;
		END_IF;
		// stNetwork - bRoleInNetwork [BOOL] [READ_WRITE]
		IF aStatInputSelections[111] THEN
			aStatCommandQueue[nTempLoopIndex].nIndex := 88;
			aStatCommandQueue[nTempLoopIndex].nSubIndex := 1;
			aStatCommandQueue[nTempLoopIndex].nBitLength := 8;
			nTempLoopIndex := nTempLoopIndex + 1;
		END_IF;
		// stNetwork - bDeviceNoMasterHighestNo [BOOL] [READ_WRITE]
		IF aStatInputSelections[112] THEN
			aStatCommandQueue[nTempLoopIndex].nIndex := 88;
			aStatCommandQueue[nTempLoopIndex].nSubIndex := 2;
			aStatCommandQueue[nTempLoopIndex].nBitLength := 8;
			nTempLoopIndex := nTempLoopIndex + 1;
		END_IF;
		// Next step
		IF stStatLastErrorCode.nBlockError = 0 THEN
			nStatState := cSTATE_CLEAR_RECORD;
		END_IF;
	END_IF;
// Clear IO-Link record
	IF nStatState = cSTATE_CLEAR_RECORD THEN
		IF bStatRWSave THEN
			FOR nTempLoopIndex := 0 TO cNUMBER_IOLINK_DATA DO
				aStatIOLRecords[nTempLoopIndex] := 16#00;
			END_FOR;
		END_IF;
		// Next step
		nStatState := cSTATE_SEND_REQUEST;
	END_IF;
// Send telegram
	IF nStatState = cSTATE_SEND_REQUEST AND NOT fbReadWriteReq.bBusy AND bStatBusyMem THEN
		CASE aStatCommandQueue[nStatCommandIndex].nIndex OF
			// stCommands [ComplexT] [WRITE_ONLY]
				32767:
					fbReadWriteReq(bRW:= bRW, nIndex := 2, nSubIndex := 0, nLen := aStatCommandQueue[nStatCommandIndex].nBitLength, aData := aStatIOLRecords);
					nStatComplex := cBASIC_TYPE;
					nStatBitLength := aStatCommandQueue[nStatCommandIndex].nBitLength;
					CASE aStatCommandQueue[nStatCommandIndex].nSubIndex OF
					// stCommands - nCmdRestoreFactorySettings [UINT] [WRITE_ONLY]
					1:
					nTempDeviceDataInteger := UINT_TO_DWORD(stDeviceData.stData.stCommands.nCmdRestoreFactorySettings);
					JMP SetInteger;
					// stCommands - nCmdTeachApply [UINT] [WRITE_ONLY]
					2:
					nTempDeviceDataInteger := UINT_TO_DWORD(stDeviceData.stData.stCommands.nCmdTeachApply);
					JMP SetInteger;
					// stCommands - nCmdSetpoint1SingleValueTeach [UINT] [WRITE_ONLY]
					3:
					nTempDeviceDataInteger := UINT_TO_DWORD(stDeviceData.stData.stCommands.nCmdSetpoint1SingleValueTeach);
					JMP SetInteger;
					// stCommands - nCmdSetpoint2SingleValueTeach [UINT] [WRITE_ONLY]
					4:
					nTempDeviceDataInteger := UINT_TO_DWORD(stDeviceData.stData.stCommands.nCmdSetpoint2SingleValueTeach);
					JMP SetInteger;
					// stCommands - nCmdTwoValueTeachTp1Sp1 [UINT] [WRITE_ONLY]
					5:
					nTempDeviceDataInteger := UINT_TO_DWORD(stDeviceData.stData.stCommands.nCmdTwoValueTeachTp1Sp1);
					JMP SetInteger;
					// stCommands - nCmdTwoValueTeachTp2Sp1 [UINT] [WRITE_ONLY]
					6:
					nTempDeviceDataInteger := UINT_TO_DWORD(stDeviceData.stData.stCommands.nCmdTwoValueTeachTp2Sp1);
					JMP SetInteger;
					// stCommands - nCmdTwoValueTeachTp1Sp2 [UINT] [WRITE_ONLY]
					7:
					nTempDeviceDataInteger := UINT_TO_DWORD(stDeviceData.stData.stCommands.nCmdTwoValueTeachTp1Sp2);
					JMP SetInteger;
					// stCommands - nCmdTwoValueTeachTp2Sp2 [UINT] [WRITE_ONLY]
					8:
					nTempDeviceDataInteger := UINT_TO_DWORD(stDeviceData.stData.stCommands.nCmdTwoValueTeachTp2Sp2);
					JMP SetInteger;
					// stCommands - nCmdSetpoint1DynamicTeachStart [UINT] [WRITE_ONLY]
					9:
					nTempDeviceDataInteger := UINT_TO_DWORD(stDeviceData.stData.stCommands.nCmdSetpoint1DynamicTeachStart);
					JMP SetInteger;
					// stCommands - nCmdSetpoint1DynamicTeachStop [UINT] [WRITE_ONLY]
					10:
					nTempDeviceDataInteger := UINT_TO_DWORD(stDeviceData.stData.stCommands.nCmdSetpoint1DynamicTeachStop);
					JMP SetInteger;
					// stCommands - nCmdSetpoint2DynamicTeachStart [UINT] [WRITE_ONLY]
					11:
					nTempDeviceDataInteger := UINT_TO_DWORD(stDeviceData.stData.stCommands.nCmdSetpoint2DynamicTeachStart);
					JMP SetInteger;
					// stCommands - nCmdSetpoint2DynamicTeachStop [UINT] [WRITE_ONLY]
					12:
					nTempDeviceDataInteger := UINT_TO_DWORD(stDeviceData.stData.stCommands.nCmdSetpoint2DynamicTeachStop);
					JMP SetInteger;
					// stCommands - nCmdTeachCancel [UINT] [WRITE_ONLY]
					13:
					nTempDeviceDataInteger := UINT_TO_DWORD(stDeviceData.stData.stCommands.nCmdTeachCancel);
					JMP SetInteger;
					// stCommands - nCmdSetAnalogOutputLowerLimit [UINT] [WRITE_ONLY]
					14:
					nTempDeviceDataInteger := UINT_TO_DWORD(stDeviceData.stData.stCommands.nCmdSetAnalogOutputLowerLimit);
					JMP SetInteger;
					// stCommands - nCmdSetAnalogOutputUpperLimit [UINT] [WRITE_ONLY]
					15:
					nTempDeviceDataInteger := UINT_TO_DWORD(stDeviceData.stData.stCommands.nCmdSetAnalogOutputUpperLimit);
					JMP SetInteger;
					// stCommands - nCmdResetDiagnosisInformation [UINT] [WRITE_ONLY]
					16:
					nTempDeviceDataInteger := UINT_TO_DWORD(stDeviceData.stData.stCommands.nCmdResetDiagnosisInformation);
					JMP SetInteger;
					// stCommands - nCmdStopMeasurement [UINT] [WRITE_ONLY]
					17:
					nTempDeviceDataInteger := UINT_TO_DWORD(stDeviceData.stData.stCommands.nCmdStopMeasurement);
					JMP SetInteger;
					// stCommands - nCmdStartMeasurement [UINT] [WRITE_ONLY]
					18:
					nTempDeviceDataInteger := UINT_TO_DWORD(stDeviceData.stData.stCommands.nCmdStartMeasurement);
					JMP SetInteger;
					// stCommands - nCmdSingleMeasurement [UINT] [WRITE_ONLY]
					19:
					nTempDeviceDataInteger := UINT_TO_DWORD(stDeviceData.stData.stCommands.nCmdSingleMeasurement);
					JMP SetInteger;
					// stCommands - nCmdIoLink11SystemTestCommand240Event8DfeAppears [UINT] [WRITE_ONLY]
					20:
					nTempDeviceDataInteger := UINT_TO_DWORD(stDeviceData.stData.stCommands.nCmdIoLink11SystemTestCommand240Event8DfeAppears);
					JMP SetInteger;
					// stCommands - nCmdIoLink11SystemTestCommand241Event8DfeDisappears [UINT] [WRITE_ONLY]
					21:
					nTempDeviceDataInteger := UINT_TO_DWORD(stDeviceData.stData.stCommands.nCmdIoLink11SystemTestCommand241Event8DfeDisappears);
					JMP SetInteger;
					// stCommands - nCmdIoLink11SystemTestCommand242Event8DffAppears [UINT] [WRITE_ONLY]
					22:
					nTempDeviceDataInteger := UINT_TO_DWORD(stDeviceData.stData.stCommands.nCmdIoLink11SystemTestCommand242Event8DffAppears);
					JMP SetInteger;
					// stCommands - nCmdIoLink11SystemTestCommand243Event8DffDisappears [UINT] [WRITE_ONLY]
					23:
					nTempDeviceDataInteger := UINT_TO_DWORD(stDeviceData.stData.stCommands.nCmdIoLink11SystemTestCommand243Event8DffDisappears);
					JMP SetInteger;
				END_CASE;
			// stDirectParametersPage1 [ComplexT] [READ_WRITE]
				0:
					fbReadWriteReq(bRW:= bRW, nIndex := aStatCommandQueue[nStatCommandIndex].nIndex, nSubIndex := aStatCommandQueue[nStatCommandIndex].nSubIndex, nLen := aStatCommandQueue[nStatCommandIndex].nBitLength, aData := aStatIOLRecords);
					IF bStatRWSave THEN
						nStatComplex := cCOMPLEX_RECORD_TYPE;
						nStatComplexDataTypeSize := UINT_TO_INT(aStatCommandQueue[nStatCommandIndex].nBitLength);
						nStatOffset := 0;
					// stDirectParametersPage1 - nSystemCommand [UINT] [WRITE_ONLY]
					IF (aStatCommandQueue[nStatCommandIndex].nSubIndex = 0 AND nStatIndex = 0) OR (aStatCommandQueue[nStatCommandIndex].nSubIndex = 16 AND nStatIndex = 0) THEN
						IF aStatCommandQueue[nStatCommandIndex].nSubIndex = 0 THEN
							  nStatOffset := 0;
						END_IF;
							nStatBitLength := 8;
							nTempDeviceDataInteger := UINT_TO_DWORD(stDeviceData.stData.stDirectParametersPage1.nSystemCommand);
							JMP SetInteger;
						END_IF;
					END_IF;
			// stDirectParametersPage2 [ComplexT] [READ_WRITE]
				1:
					fbReadWriteReq(bRW:= bRW, nIndex := aStatCommandQueue[nStatCommandIndex].nIndex, nSubIndex := aStatCommandQueue[nStatCommandIndex].nSubIndex, nLen := aStatCommandQueue[nStatCommandIndex].nBitLength, aData := aStatIOLRecords);
					IF bStatRWSave THEN
						nStatComplex := cCOMPLEX_RECORD_TYPE;
						nStatComplexDataTypeSize := UINT_TO_INT(aStatCommandQueue[nStatCommandIndex].nBitLength);
						nStatOffset := 0;
					// stDirectParametersPage2 - nDeviceSpecificParameter1 [UINT] [READ_WRITE]
					IF (aStatCommandQueue[nStatCommandIndex].nSubIndex = 0 AND nStatIndex = 0) OR (aStatCommandQueue[nStatCommandIndex].nSubIndex = 1 AND nStatIndex = 0) THEN
						IF aStatCommandQueue[nStatCommandIndex].nSubIndex = 0 THEN
							  nStatOffset := 120;
						END_IF;
							nStatBitLength := 8;
							nTempDeviceDataInteger := UINT_TO_DWORD(stDeviceData.stData.stDirectParametersPage2.nDeviceSpecificParameter1);
							JMP SetInteger;
						END_IF;
					// stDirectParametersPage2 - nDeviceSpecificParameter2 [UINT] [READ_WRITE]
					IF (aStatCommandQueue[nStatCommandIndex].nSubIndex = 0 AND nStatIndex = 1) OR (aStatCommandQueue[nStatCommandIndex].nSubIndex = 2 AND nStatIndex = 0) THEN
						IF aStatCommandQueue[nStatCommandIndex].nSubIndex = 0 THEN
							  nStatOffset := 112;
						END_IF;
							nStatBitLength := 8;
							nTempDeviceDataInteger := UINT_TO_DWORD(stDeviceData.stData.stDirectParametersPage2.nDeviceSpecificParameter2);
							JMP SetInteger;
						END_IF;
					// stDirectParametersPage2 - nDeviceSpecificParameter3 [UINT] [READ_WRITE]
					IF (aStatCommandQueue[nStatCommandIndex].nSubIndex = 0 AND nStatIndex = 2) OR (aStatCommandQueue[nStatCommandIndex].nSubIndex = 3 AND nStatIndex = 0) THEN
						IF aStatCommandQueue[nStatCommandIndex].nSubIndex = 0 THEN
							  nStatOffset := 104;
						END_IF;
							nStatBitLength := 8;
							nTempDeviceDataInteger := UINT_TO_DWORD(stDeviceData.stData.stDirectParametersPage2.nDeviceSpecificParameter3);
							JMP SetInteger;
						END_IF;
					// stDirectParametersPage2 - nDeviceSpecificParameter4 [UINT] [READ_WRITE]
					IF (aStatCommandQueue[nStatCommandIndex].nSubIndex = 0 AND nStatIndex = 3) OR (aStatCommandQueue[nStatCommandIndex].nSubIndex = 4 AND nStatIndex = 0) THEN
						IF aStatCommandQueue[nStatCommandIndex].nSubIndex = 0 THEN
							  nStatOffset := 96;
						END_IF;
							nStatBitLength := 8;
							nTempDeviceDataInteger := UINT_TO_DWORD(stDeviceData.stData.stDirectParametersPage2.nDeviceSpecificParameter4);
							JMP SetInteger;
						END_IF;
					// stDirectParametersPage2 - nDeviceSpecificParameter5 [UINT] [READ_WRITE]
					IF (aStatCommandQueue[nStatCommandIndex].nSubIndex = 0 AND nStatIndex = 4) OR (aStatCommandQueue[nStatCommandIndex].nSubIndex = 5 AND nStatIndex = 0) THEN
						IF aStatCommandQueue[nStatCommandIndex].nSubIndex = 0 THEN
							  nStatOffset := 88;
						END_IF;
							nStatBitLength := 8;
							nTempDeviceDataInteger := UINT_TO_DWORD(stDeviceData.stData.stDirectParametersPage2.nDeviceSpecificParameter5);
							JMP SetInteger;
						END_IF;
					// stDirectParametersPage2 - nDeviceSpecificParameter6 [UINT] [READ_WRITE]
					IF (aStatCommandQueue[nStatCommandIndex].nSubIndex = 0 AND nStatIndex = 5) OR (aStatCommandQueue[nStatCommandIndex].nSubIndex = 6 AND nStatIndex = 0) THEN
						IF aStatCommandQueue[nStatCommandIndex].nSubIndex = 0 THEN
							  nStatOffset := 80;
						END_IF;
							nStatBitLength := 8;
							nTempDeviceDataInteger := UINT_TO_DWORD(stDeviceData.stData.stDirectParametersPage2.nDeviceSpecificParameter6);
							JMP SetInteger;
						END_IF;
					// stDirectParametersPage2 - nDeviceSpecificParameter7 [UINT] [READ_WRITE]
					IF (aStatCommandQueue[nStatCommandIndex].nSubIndex = 0 AND nStatIndex = 6) OR (aStatCommandQueue[nStatCommandIndex].nSubIndex = 7 AND nStatIndex = 0) THEN
						IF aStatCommandQueue[nStatCommandIndex].nSubIndex = 0 THEN
							  nStatOffset := 72;
						END_IF;
							nStatBitLength := 8;
							nTempDeviceDataInteger := UINT_TO_DWORD(stDeviceData.stData.stDirectParametersPage2.nDeviceSpecificParameter7);
							JMP SetInteger;
						END_IF;
					// stDirectParametersPage2 - nDeviceSpecificParameter8 [UINT] [READ_WRITE]
					IF (aStatCommandQueue[nStatCommandIndex].nSubIndex = 0 AND nStatIndex = 7) OR (aStatCommandQueue[nStatCommandIndex].nSubIndex = 8 AND nStatIndex = 0) THEN
						IF aStatCommandQueue[nStatCommandIndex].nSubIndex = 0 THEN
							  nStatOffset := 64;
						END_IF;
							nStatBitLength := 8;
							nTempDeviceDataInteger := UINT_TO_DWORD(stDeviceData.stData.stDirectParametersPage2.nDeviceSpecificParameter8);
							JMP SetInteger;
						END_IF;
					// stDirectParametersPage2 - nDeviceSpecificParameter9 [UINT] [READ_WRITE]
					IF (aStatCommandQueue[nStatCommandIndex].nSubIndex = 0 AND nStatIndex = 8) OR (aStatCommandQueue[nStatCommandIndex].nSubIndex = 9 AND nStatIndex = 0) THEN
						IF aStatCommandQueue[nStatCommandIndex].nSubIndex = 0 THEN
							  nStatOffset := 56;
						END_IF;
							nStatBitLength := 8;
							nTempDeviceDataInteger := UINT_TO_DWORD(stDeviceData.stData.stDirectParametersPage2.nDeviceSpecificParameter9);
							JMP SetInteger;
						END_IF;
					// stDirectParametersPage2 - nDeviceSpecificParameter10 [UINT] [READ_WRITE]
					IF (aStatCommandQueue[nStatCommandIndex].nSubIndex = 0 AND nStatIndex = 9) OR (aStatCommandQueue[nStatCommandIndex].nSubIndex = 10 AND nStatIndex = 0) THEN
						IF aStatCommandQueue[nStatCommandIndex].nSubIndex = 0 THEN
							  nStatOffset := 48;
						END_IF;
							nStatBitLength := 8;
							nTempDeviceDataInteger := UINT_TO_DWORD(stDeviceData.stData.stDirectParametersPage2.nDeviceSpecificParameter10);
							JMP SetInteger;
						END_IF;
					// stDirectParametersPage2 - nDeviceSpecificParameter11 [UINT] [READ_WRITE]
					IF (aStatCommandQueue[nStatCommandIndex].nSubIndex = 0 AND nStatIndex = 10) OR (aStatCommandQueue[nStatCommandIndex].nSubIndex = 11 AND nStatIndex = 0) THEN
						IF aStatCommandQueue[nStatCommandIndex].nSubIndex = 0 THEN
							  nStatOffset := 40;
						END_IF;
							nStatBitLength := 8;
							nTempDeviceDataInteger := UINT_TO_DWORD(stDeviceData.stData.stDirectParametersPage2.nDeviceSpecificParameter11);
							JMP SetInteger;
						END_IF;
					// stDirectParametersPage2 - nDeviceSpecificParameter12 [UINT] [READ_WRITE]
					IF (aStatCommandQueue[nStatCommandIndex].nSubIndex = 0 AND nStatIndex = 11) OR (aStatCommandQueue[nStatCommandIndex].nSubIndex = 12 AND nStatIndex = 0) THEN
						IF aStatCommandQueue[nStatCommandIndex].nSubIndex = 0 THEN
							  nStatOffset := 32;
						END_IF;
							nStatBitLength := 8;
							nTempDeviceDataInteger := UINT_TO_DWORD(stDeviceData.stData.stDirectParametersPage2.nDeviceSpecificParameter12);
							JMP SetInteger;
						END_IF;
					// stDirectParametersPage2 - nDeviceSpecificParameter13 [UINT] [READ_WRITE]
					IF (aStatCommandQueue[nStatCommandIndex].nSubIndex = 0 AND nStatIndex = 12) OR (aStatCommandQueue[nStatCommandIndex].nSubIndex = 13 AND nStatIndex = 0) THEN
						IF aStatCommandQueue[nStatCommandIndex].nSubIndex = 0 THEN
							  nStatOffset := 24;
						END_IF;
							nStatBitLength := 8;
							nTempDeviceDataInteger := UINT_TO_DWORD(stDeviceData.stData.stDirectParametersPage2.nDeviceSpecificParameter13);
							JMP SetInteger;
						END_IF;
					// stDirectParametersPage2 - nDeviceSpecificParameter14 [UINT] [READ_WRITE]
					IF (aStatCommandQueue[nStatCommandIndex].nSubIndex = 0 AND nStatIndex = 13) OR (aStatCommandQueue[nStatCommandIndex].nSubIndex = 14 AND nStatIndex = 0) THEN
						IF aStatCommandQueue[nStatCommandIndex].nSubIndex = 0 THEN
							  nStatOffset := 16;
						END_IF;
							nStatBitLength := 8;
							nTempDeviceDataInteger := UINT_TO_DWORD(stDeviceData.stData.stDirectParametersPage2.nDeviceSpecificParameter14);
							JMP SetInteger;
						END_IF;
					// stDirectParametersPage2 - nDeviceSpecificParameter15 [UINT] [READ_WRITE]
					IF (aStatCommandQueue[nStatCommandIndex].nSubIndex = 0 AND nStatIndex = 14) OR (aStatCommandQueue[nStatCommandIndex].nSubIndex = 15 AND nStatIndex = 0) THEN
						IF aStatCommandQueue[nStatCommandIndex].nSubIndex = 0 THEN
							  nStatOffset := 8;
						END_IF;
							nStatBitLength := 8;
							nTempDeviceDataInteger := UINT_TO_DWORD(stDeviceData.stData.stDirectParametersPage2.nDeviceSpecificParameter15);
							JMP SetInteger;
						END_IF;
					// stDirectParametersPage2 - nDeviceSpecificParameter16 [UINT] [READ_WRITE]
					IF (aStatCommandQueue[nStatCommandIndex].nSubIndex = 0 AND nStatIndex = 15) OR (aStatCommandQueue[nStatCommandIndex].nSubIndex = 16 AND nStatIndex = 0) THEN
						IF aStatCommandQueue[nStatCommandIndex].nSubIndex = 0 THEN
							  nStatOffset := 0;
						END_IF;
							nStatBitLength := 8;
							nTempDeviceDataInteger := UINT_TO_DWORD(stDeviceData.stData.stDirectParametersPage2.nDeviceSpecificParameter16);
							JMP SetInteger;
						END_IF;
					END_IF;
			// nSystemCommand [UINT] [WRITE_ONLY]
				2:
					fbReadWriteReq(bRW:= bRW, nIndex := aStatCommandQueue[nStatCommandIndex].nIndex, nSubIndex := aStatCommandQueue[nStatCommandIndex].nSubIndex, nLen := aStatCommandQueue[nStatCommandIndex].nBitLength, aData := aStatIOLRecords);
					IF bStatRWSave THEN
						nStatComplex := cBASIC_TYPE;
						nStatBitLength := aStatCommandQueue[nStatCommandIndex].nBitLength;
						nTempDeviceDataInteger := UINT_TO_DWORD(stDeviceData.stData.nSystemCommand);
						JMP SetInteger;
					END_IF;
			// stDeviceAccessLocks [ComplexT] [READ_WRITE]
				12:
					fbReadWriteReq(bRW:= bRW, nIndex := aStatCommandQueue[nStatCommandIndex].nIndex, nSubIndex := aStatCommandQueue[nStatCommandIndex].nSubIndex, nLen := aStatCommandQueue[nStatCommandIndex].nBitLength, aData := aStatIOLRecords);
					IF bStatRWSave THEN
						nStatComplex := cCOMPLEX_RECORD_TYPE;
						nStatComplexDataTypeSize := UINT_TO_INT(aStatCommandQueue[nStatCommandIndex].nBitLength);
						nStatOffset := 0;
					// stDeviceAccessLocks - bParameterWriteAccess [BOOL] [READ_WRITE]
						IF (aStatCommandQueue[nStatCommandIndex].nSubIndex = 0 AND nStatIndex = 0) THEN
							nStatOffset := 0;
							bTempDeviceDataBool := stDeviceData.stData.stDeviceAccessLocks.bParameterWriteAccess;
							JMP SetBoolean;
						END_IF;
					// stDeviceAccessLocks - bDataStorage [BOOL] [READ_WRITE]
						IF (aStatCommandQueue[nStatCommandIndex].nSubIndex = 0 AND nStatIndex = 1) THEN
							nStatOffset := 1;
							bTempDeviceDataBool := stDeviceData.stData.stDeviceAccessLocks.bDataStorage;
							JMP SetBoolean;
						END_IF;
					// stDeviceAccessLocks - bLocalParameterization [BOOL] [READ_WRITE]
						IF (aStatCommandQueue[nStatCommandIndex].nSubIndex = 0 AND nStatIndex = 2) THEN
							nStatOffset := 2;
							bTempDeviceDataBool := stDeviceData.stData.stDeviceAccessLocks.bLocalParameterization;
							JMP SetBoolean;
						END_IF;
					// stDeviceAccessLocks - bLocalUserInterface [BOOL] [READ_WRITE]
						IF (aStatCommandQueue[nStatCommandIndex].nSubIndex = 0 AND nStatIndex = 3) THEN
							nStatOffset := 3;
							bTempDeviceDataBool := stDeviceData.stData.stDeviceAccessLocks.bLocalUserInterface;
							JMP SetBoolean;
						END_IF;
					END_IF;
			// sVendorName [STRING] [READ_ONLY]
				16:
					fbReadWriteReq(bRW:= bRW, nIndex := aStatCommandQueue[nStatCommandIndex].nIndex, nSubIndex := aStatCommandQueue[nStatCommandIndex].nSubIndex, nLen := aStatCommandQueue[nStatCommandIndex].nBitLength, aData := aStatIOLRecords);
			// sVendorText [STRING] [READ_ONLY]
				17:
					fbReadWriteReq(bRW:= bRW, nIndex := aStatCommandQueue[nStatCommandIndex].nIndex, nSubIndex := aStatCommandQueue[nStatCommandIndex].nSubIndex, nLen := aStatCommandQueue[nStatCommandIndex].nBitLength, aData := aStatIOLRecords);
			// sProductName [STRING] [READ_ONLY]
				18:
					fbReadWriteReq(bRW:= bRW, nIndex := aStatCommandQueue[nStatCommandIndex].nIndex, nSubIndex := aStatCommandQueue[nStatCommandIndex].nSubIndex, nLen := aStatCommandQueue[nStatCommandIndex].nBitLength, aData := aStatIOLRecords);
			// sProductId [STRING] [READ_ONLY]
				19:
					fbReadWriteReq(bRW:= bRW, nIndex := aStatCommandQueue[nStatCommandIndex].nIndex, nSubIndex := aStatCommandQueue[nStatCommandIndex].nSubIndex, nLen := aStatCommandQueue[nStatCommandIndex].nBitLength, aData := aStatIOLRecords);
			// sProductText [STRING] [READ_ONLY]
				20:
					fbReadWriteReq(bRW:= bRW, nIndex := aStatCommandQueue[nStatCommandIndex].nIndex, nSubIndex := aStatCommandQueue[nStatCommandIndex].nSubIndex, nLen := aStatCommandQueue[nStatCommandIndex].nBitLength, aData := aStatIOLRecords);
			// sFirmwareRevision [STRING] [READ_ONLY]
				23:
					fbReadWriteReq(bRW:= bRW, nIndex := aStatCommandQueue[nStatCommandIndex].nIndex, nSubIndex := aStatCommandQueue[nStatCommandIndex].nSubIndex, nLen := aStatCommandQueue[nStatCommandIndex].nBitLength, aData := aStatIOLRecords);
			// sApplicationSpecificTag [STRING] [READ_WRITE]
				24:
					fbReadWriteReq(bRW:= bRW, nIndex := aStatCommandQueue[nStatCommandIndex].nIndex, nSubIndex := aStatCommandQueue[nStatCommandIndex].nSubIndex, nLen := aStatCommandQueue[nStatCommandIndex].nBitLength, aData := aStatIOLRecords);
					IF bStatRWSave THEN
						nStatComplex := cBASIC_TYPE;
						nStatBitLength := aStatCommandQueue[nStatCommandIndex].nBitLength;
						sTempDeviceDataString := stDeviceData.stData.sApplicationSpecificTag;
						JMP SetString;
					END_IF;
			// nErrorCount [UINT] [READ_ONLY]
				32:
					fbReadWriteReq(bRW:= bRW, nIndex := aStatCommandQueue[nStatCommandIndex].nIndex, nSubIndex := aStatCommandQueue[nStatCommandIndex].nSubIndex, nLen := aStatCommandQueue[nStatCommandIndex].nBitLength, aData := aStatIOLRecords);
			// nDeviceStatus [UINT] [READ_ONLY]
				36:
					fbReadWriteReq(bRW:= bRW, nIndex := aStatCommandQueue[nStatCommandIndex].nIndex, nSubIndex := aStatCommandQueue[nStatCommandIndex].nSubIndex, nLen := aStatCommandQueue[nStatCommandIndex].nBitLength, aData := aStatIOLRecords);
			// nTeachInSelect [UINT] [READ_WRITE]
				58:
					fbReadWriteReq(bRW:= bRW, nIndex := aStatCommandQueue[nStatCommandIndex].nIndex, nSubIndex := aStatCommandQueue[nStatCommandIndex].nSubIndex, nLen := aStatCommandQueue[nStatCommandIndex].nBitLength, aData := aStatIOLRecords);
					IF bStatRWSave THEN
						nStatComplex := cBASIC_TYPE;
						nStatBitLength := aStatCommandQueue[nStatCommandIndex].nBitLength;
						nTempDeviceDataInteger := UINT_TO_DWORD(stDeviceData.stData.nTeachInSelect);
						JMP SetInteger;
					END_IF;
			// stTeachState [ComplexT] [READ_ONLY]
				59:
					fbReadWriteReq(bRW:= bRW, nIndex := aStatCommandQueue[nStatCommandIndex].nIndex, nSubIndex := aStatCommandQueue[nStatCommandIndex].nSubIndex, nLen := aStatCommandQueue[nStatCommandIndex].nBitLength, aData := aStatIOLRecords);
			// stSetpoints_60 [ComplexT] [READ_WRITE]
				60:
					fbReadWriteReq(bRW:= bRW, nIndex := aStatCommandQueue[nStatCommandIndex].nIndex, nSubIndex := aStatCommandQueue[nStatCommandIndex].nSubIndex, nLen := aStatCommandQueue[nStatCommandIndex].nBitLength, aData := aStatIOLRecords);
					IF bStatRWSave THEN
						nStatComplex := cCOMPLEX_RECORD_TYPE;
						nStatComplexDataTypeSize := UINT_TO_INT(aStatCommandQueue[nStatCommandIndex].nBitLength);
						nStatOffset := 0;
					// stSetpoints_60 - nParam1Bdc1Q1 [UINT] [READ_WRITE]
					IF (aStatCommandQueue[nStatCommandIndex].nSubIndex = 0 AND nStatIndex = 0) OR (aStatCommandQueue[nStatCommandIndex].nSubIndex = 1 AND nStatIndex = 0) THEN
						IF aStatCommandQueue[nStatCommandIndex].nSubIndex = 0 THEN
							  nStatOffset := 16;
						END_IF;
							nStatBitLength := 16;
							nTempDeviceDataInteger := UINT_TO_DWORD(stDeviceData.stData.stSetpoints_60.nParam1Bdc1Q1);
							JMP SetInteger;
						END_IF;
					// stSetpoints_60 - nParam2Bdc1Q1 [UINT] [READ_WRITE]
					IF (aStatCommandQueue[nStatCommandIndex].nSubIndex = 0 AND nStatIndex = 1) OR (aStatCommandQueue[nStatCommandIndex].nSubIndex = 2 AND nStatIndex = 0) THEN
						IF aStatCommandQueue[nStatCommandIndex].nSubIndex = 0 THEN
							  nStatOffset := 0;
						END_IF;
							nStatBitLength := 16;
							nTempDeviceDataInteger := UINT_TO_DWORD(stDeviceData.stData.stSetpoints_60.nParam2Bdc1Q1);
							JMP SetInteger;
						END_IF;
					END_IF;
			// stSwitchpointBdc1 [ComplexT] [READ_WRITE]
				61:
					fbReadWriteReq(bRW:= bRW, nIndex := aStatCommandQueue[nStatCommandIndex].nIndex, nSubIndex := aStatCommandQueue[nStatCommandIndex].nSubIndex, nLen := aStatCommandQueue[nStatCommandIndex].nBitLength, aData := aStatIOLRecords);
					IF bStatRWSave THEN
						nStatComplex := cCOMPLEX_RECORD_TYPE;
						nStatComplexDataTypeSize := UINT_TO_INT(aStatCommandQueue[nStatCommandIndex].nBitLength);
						nStatOffset := 0;
					// stSwitchpointBdc1 - nLogic [UINT] [READ_WRITE]
					IF (aStatCommandQueue[nStatCommandIndex].nSubIndex = 0 AND nStatIndex = 0) OR (aStatCommandQueue[nStatCommandIndex].nSubIndex = 1 AND nStatIndex = 0) THEN
						IF aStatCommandQueue[nStatCommandIndex].nSubIndex = 0 THEN
							  nStatOffset := 24;
						END_IF;
							nStatBitLength := 8;
							nTempDeviceDataInteger := UINT_TO_DWORD(stDeviceData.stData.stSwitchpointBdc1.nLogic);
							JMP SetInteger;
						END_IF;
					// stSwitchpointBdc1 - nMode [UINT] [READ_WRITE]
					IF (aStatCommandQueue[nStatCommandIndex].nSubIndex = 0 AND nStatIndex = 1) OR (aStatCommandQueue[nStatCommandIndex].nSubIndex = 2 AND nStatIndex = 0) THEN
						IF aStatCommandQueue[nStatCommandIndex].nSubIndex = 0 THEN
							  nStatOffset := 16;
						END_IF;
							nStatBitLength := 8;
							nTempDeviceDataInteger := UINT_TO_DWORD(stDeviceData.stData.stSwitchpointBdc1.nMode);
							JMP SetInteger;
						END_IF;
					// stSwitchpointBdc1 - nHysteresis [UINT] [READ_WRITE]
					IF (aStatCommandQueue[nStatCommandIndex].nSubIndex = 0 AND nStatIndex = 2) OR (aStatCommandQueue[nStatCommandIndex].nSubIndex = 3 AND nStatIndex = 0) THEN
						IF aStatCommandQueue[nStatCommandIndex].nSubIndex = 0 THEN
							  nStatOffset := 0;
						END_IF;
							nStatBitLength := 16;
							nTempDeviceDataInteger := UINT_TO_DWORD(stDeviceData.stData.stSwitchpointBdc1.nHysteresis);
							JMP SetInteger;
						END_IF;
					END_IF;
			// stSetpoints_62 [ComplexT] [READ_WRITE]
				62:
					fbReadWriteReq(bRW:= bRW, nIndex := aStatCommandQueue[nStatCommandIndex].nIndex, nSubIndex := aStatCommandQueue[nStatCommandIndex].nSubIndex, nLen := aStatCommandQueue[nStatCommandIndex].nBitLength, aData := aStatIOLRecords);
					IF bStatRWSave THEN
						nStatComplex := cCOMPLEX_RECORD_TYPE;
						nStatComplexDataTypeSize := UINT_TO_INT(aStatCommandQueue[nStatCommandIndex].nBitLength);
						nStatOffset := 0;
					// stSetpoints_62 - nParam1Bdc2Q2 [UINT] [READ_WRITE]
					IF (aStatCommandQueue[nStatCommandIndex].nSubIndex = 0 AND nStatIndex = 0) OR (aStatCommandQueue[nStatCommandIndex].nSubIndex = 1 AND nStatIndex = 0) THEN
						IF aStatCommandQueue[nStatCommandIndex].nSubIndex = 0 THEN
							  nStatOffset := 16;
						END_IF;
							nStatBitLength := 16;
							nTempDeviceDataInteger := UINT_TO_DWORD(stDeviceData.stData.stSetpoints_62.nParam1Bdc2Q2);
							JMP SetInteger;
						END_IF;
					// stSetpoints_62 - nParam2Bdc2Q2 [UINT] [READ_WRITE]
					IF (aStatCommandQueue[nStatCommandIndex].nSubIndex = 0 AND nStatIndex = 1) OR (aStatCommandQueue[nStatCommandIndex].nSubIndex = 2 AND nStatIndex = 0) THEN
						IF aStatCommandQueue[nStatCommandIndex].nSubIndex = 0 THEN
							  nStatOffset := 0;
						END_IF;
							nStatBitLength := 16;
							nTempDeviceDataInteger := UINT_TO_DWORD(stDeviceData.stData.stSetpoints_62.nParam2Bdc2Q2);
							JMP SetInteger;
						END_IF;
					END_IF;
			// stSwitchpointBdc2 [ComplexT] [READ_WRITE]
				63:
					fbReadWriteReq(bRW:= bRW, nIndex := aStatCommandQueue[nStatCommandIndex].nIndex, nSubIndex := aStatCommandQueue[nStatCommandIndex].nSubIndex, nLen := aStatCommandQueue[nStatCommandIndex].nBitLength, aData := aStatIOLRecords);
					IF bStatRWSave THEN
						nStatComplex := cCOMPLEX_RECORD_TYPE;
						nStatComplexDataTypeSize := UINT_TO_INT(aStatCommandQueue[nStatCommandIndex].nBitLength);
						nStatOffset := 0;
					// stSwitchpointBdc2 - nLogic [UINT] [READ_WRITE]
					IF (aStatCommandQueue[nStatCommandIndex].nSubIndex = 0 AND nStatIndex = 0) OR (aStatCommandQueue[nStatCommandIndex].nSubIndex = 1 AND nStatIndex = 0) THEN
						IF aStatCommandQueue[nStatCommandIndex].nSubIndex = 0 THEN
							  nStatOffset := 24;
						END_IF;
							nStatBitLength := 8;
							nTempDeviceDataInteger := UINT_TO_DWORD(stDeviceData.stData.stSwitchpointBdc2.nLogic);
							JMP SetInteger;
						END_IF;
					// stSwitchpointBdc2 - nMode [UINT] [READ_WRITE]
					IF (aStatCommandQueue[nStatCommandIndex].nSubIndex = 0 AND nStatIndex = 1) OR (aStatCommandQueue[nStatCommandIndex].nSubIndex = 2 AND nStatIndex = 0) THEN
						IF aStatCommandQueue[nStatCommandIndex].nSubIndex = 0 THEN
							  nStatOffset := 16;
						END_IF;
							nStatBitLength := 8;
							nTempDeviceDataInteger := UINT_TO_DWORD(stDeviceData.stData.stSwitchpointBdc2.nMode);
							JMP SetInteger;
						END_IF;
					// stSwitchpointBdc2 - nHysteresis [UINT] [READ_WRITE]
					IF (aStatCommandQueue[nStatCommandIndex].nSubIndex = 0 AND nStatIndex = 2) OR (aStatCommandQueue[nStatCommandIndex].nSubIndex = 3 AND nStatIndex = 0) THEN
						IF aStatCommandQueue[nStatCommandIndex].nSubIndex = 0 THEN
							  nStatOffset := 0;
						END_IF;
							nStatBitLength := 16;
							nTempDeviceDataInteger := UINT_TO_DWORD(stDeviceData.stData.stSwitchpointBdc2.nHysteresis);
							JMP SetInteger;
						END_IF;
					END_IF;
			// sLot [STRING] [READ_ONLY]
				64:
					fbReadWriteReq(bRW:= bRW, nIndex := aStatCommandQueue[nStatCommandIndex].nIndex, nSubIndex := aStatCommandQueue[nStatCommandIndex].nSubIndex, nLen := aStatCommandQueue[nStatCommandIndex].nBitLength, aData := aStatIOLRecords);
			// nOnDelaySwitchingOutput [UINT] [READ_WRITE]
				66:
					fbReadWriteReq(bRW:= bRW, nIndex := aStatCommandQueue[nStatCommandIndex].nIndex, nSubIndex := aStatCommandQueue[nStatCommandIndex].nSubIndex, nLen := aStatCommandQueue[nStatCommandIndex].nBitLength, aData := aStatIOLRecords);
					IF bStatRWSave THEN
						nStatComplex := cBASIC_TYPE;
						nStatBitLength := aStatCommandQueue[nStatCommandIndex].nBitLength;
						nTempDeviceDataInteger := UINT_TO_DWORD(stDeviceData.stData.nOnDelaySwitchingOutput);
						JMP SetInteger;
					END_IF;
			// nOffDelaySwitchingOutput [UINT] [READ_WRITE]
				67:
					fbReadWriteReq(bRW:= bRW, nIndex := aStatCommandQueue[nStatCommandIndex].nIndex, nSubIndex := aStatCommandQueue[nStatCommandIndex].nSubIndex, nLen := aStatCommandQueue[nStatCommandIndex].nBitLength, aData := aStatIOLRecords);
					IF bStatRWSave THEN
						nStatComplex := cBASIC_TYPE;
						nStatBitLength := aStatCommandQueue[nStatCommandIndex].nBitLength;
						nTempDeviceDataInteger := UINT_TO_DWORD(stDeviceData.stData.nOffDelaySwitchingOutput);
						JMP SetInteger;
					END_IF;
			// nMultiIOPin4 [UINT] [READ_WRITE]
				70:
					fbReadWriteReq(bRW:= bRW, nIndex := aStatCommandQueue[nStatCommandIndex].nIndex, nSubIndex := aStatCommandQueue[nStatCommandIndex].nSubIndex, nLen := aStatCommandQueue[nStatCommandIndex].nBitLength, aData := aStatIOLRecords);
					IF bStatRWSave THEN
						nStatComplex := cBASIC_TYPE;
						nStatBitLength := aStatCommandQueue[nStatCommandIndex].nBitLength;
						nTempDeviceDataInteger := UINT_TO_DWORD(stDeviceData.stData.nMultiIOPin4);
						JMP SetInteger;
					END_IF;
			// nMultiIOPin2 [UINT] [READ_WRITE]
				71:
					fbReadWriteReq(bRW:= bRW, nIndex := aStatCommandQueue[nStatCommandIndex].nIndex, nSubIndex := aStatCommandQueue[nStatCommandIndex].nSubIndex, nLen := aStatCommandQueue[nStatCommandIndex].nBitLength, aData := aStatIOLRecords);
					IF bStatRWSave THEN
						nStatComplex := cBASIC_TYPE;
						nStatBitLength := aStatCommandQueue[nStatCommandIndex].nBitLength;
						nTempDeviceDataInteger := UINT_TO_DWORD(stDeviceData.stData.nMultiIOPin2);
						JMP SetInteger;
					END_IF;
			// stAnalogRange [ComplexT] [READ_WRITE]
				72:
					fbReadWriteReq(bRW:= bRW, nIndex := aStatCommandQueue[nStatCommandIndex].nIndex, nSubIndex := aStatCommandQueue[nStatCommandIndex].nSubIndex, nLen := aStatCommandQueue[nStatCommandIndex].nBitLength, aData := aStatIOLRecords);
					IF bStatRWSave THEN
						nStatComplex := cCOMPLEX_RECORD_TYPE;
						nStatComplexDataTypeSize := UINT_TO_INT(aStatCommandQueue[nStatCommandIndex].nBitLength);
						nStatOffset := 0;
					// stAnalogRange - nLowerLimit [UINT] [READ_WRITE]
					IF (aStatCommandQueue[nStatCommandIndex].nSubIndex = 0 AND nStatIndex = 0) OR (aStatCommandQueue[nStatCommandIndex].nSubIndex = 1 AND nStatIndex = 0) THEN
						IF aStatCommandQueue[nStatCommandIndex].nSubIndex = 0 THEN
							  nStatOffset := 16;
						END_IF;
							nStatBitLength := 16;
							nTempDeviceDataInteger := UINT_TO_DWORD(stDeviceData.stData.stAnalogRange.nLowerLimit);
							JMP SetInteger;
						END_IF;
					// stAnalogRange - nUpperLimit [UINT] [READ_WRITE]
					IF (aStatCommandQueue[nStatCommandIndex].nSubIndex = 0 AND nStatIndex = 1) OR (aStatCommandQueue[nStatCommandIndex].nSubIndex = 2 AND nStatIndex = 0) THEN
						IF aStatCommandQueue[nStatCommandIndex].nSubIndex = 0 THEN
							  nStatOffset := 0;
						END_IF;
							nStatBitLength := 16;
							nTempDeviceDataInteger := UINT_TO_DWORD(stDeviceData.stData.stAnalogRange.nUpperLimit);
							JMP SetInteger;
						END_IF;
					END_IF;
			// nTemperatureCompensation [UINT] [READ_WRITE]
				74:
					fbReadWriteReq(bRW:= bRW, nIndex := aStatCommandQueue[nStatCommandIndex].nIndex, nSubIndex := aStatCommandQueue[nStatCommandIndex].nSubIndex, nLen := aStatCommandQueue[nStatCommandIndex].nBitLength, aData := aStatIOLRecords);
					IF bStatRWSave THEN
						nStatComplex := cBASIC_TYPE;
						nStatBitLength := aStatCommandQueue[nStatCommandIndex].nBitLength;
						nTempDeviceDataInteger := UINT_TO_DWORD(stDeviceData.stData.nTemperatureCompensation);
						JMP SetInteger;
					END_IF;
			// stTeachpointSp1_80 [ComplexT] [READ_ONLY]
				80:
					fbReadWriteReq(bRW:= bRW, nIndex := aStatCommandQueue[nStatCommandIndex].nIndex, nSubIndex := aStatCommandQueue[nStatCommandIndex].nSubIndex, nLen := aStatCommandQueue[nStatCommandIndex].nBitLength, aData := aStatIOLRecords);
			// stTeachpointSp2_81 [ComplexT] [READ_ONLY]
				81:
					fbReadWriteReq(bRW:= bRW, nIndex := aStatCommandQueue[nStatCommandIndex].nIndex, nSubIndex := aStatCommandQueue[nStatCommandIndex].nSubIndex, nLen := aStatCommandQueue[nStatCommandIndex].nBitLength, aData := aStatIOLRecords);
			// stTeachpointSp1_82 [ComplexT] [READ_ONLY]
				82:
					fbReadWriteReq(bRW:= bRW, nIndex := aStatCommandQueue[nStatCommandIndex].nIndex, nSubIndex := aStatCommandQueue[nStatCommandIndex].nSubIndex, nLen := aStatCommandQueue[nStatCommandIndex].nBitLength, aData := aStatIOLRecords);
			// stTeachpointSp2_83 [ComplexT] [READ_ONLY]
				83:
					fbReadWriteReq(bRW:= bRW, nIndex := aStatCommandQueue[nStatCommandIndex].nIndex, nSubIndex := aStatCommandQueue[nStatCommandIndex].nSubIndex, nLen := aStatCommandQueue[nStatCommandIndex].nBitLength, aData := aStatIOLRecords);
			// stProcessDataLimits [ComplexT] [READ_ONLY]
				84:
					fbReadWriteReq(bRW:= bRW, nIndex := aStatCommandQueue[nStatCommandIndex].nIndex, nSubIndex := aStatCommandQueue[nStatCommandIndex].nSubIndex, nLen := aStatCommandQueue[nStatCommandIndex].nBitLength, aData := aStatIOLRecords);
			// nSwitchCounter [UINT] [READ_ONLY]
				85:
					fbReadWriteReq(bRW:= bRW, nIndex := aStatCommandQueue[nStatCommandIndex].nIndex, nSubIndex := aStatCommandQueue[nStatCommandIndex].nSubIndex, nLen := aStatCommandQueue[nStatCommandIndex].nBitLength, aData := aStatIOLRecords);
			// nTemperatureInternal [INT] [READ_ONLY]
				86:
					fbReadWriteReq(bRW:= bRW, nIndex := aStatCommandQueue[nStatCommandIndex].nIndex, nSubIndex := aStatCommandQueue[nStatCommandIndex].nSubIndex, nLen := aStatCommandQueue[nStatCommandIndex].nBitLength, aData := aStatIOLRecords);
			// stNetwork [ComplexT] [READ_WRITE]
				88:
					fbReadWriteReq(bRW:= bRW, nIndex := aStatCommandQueue[nStatCommandIndex].nIndex, nSubIndex := aStatCommandQueue[nStatCommandIndex].nSubIndex, nLen := aStatCommandQueue[nStatCommandIndex].nBitLength, aData := aStatIOLRecords);
					IF bStatRWSave THEN
						nStatComplex := cCOMPLEX_RECORD_TYPE;
						nStatComplexDataTypeSize := UINT_TO_INT(aStatCommandQueue[nStatCommandIndex].nBitLength);
						nStatOffset := 0;
					// stNetwork - nRoleInNetwork [UINT] [READ_WRITE]
					IF (aStatCommandQueue[nStatCommandIndex].nSubIndex = 0 AND nStatIndex = 0) OR (aStatCommandQueue[nStatCommandIndex].nSubIndex = 1 AND nStatIndex = 0) THEN
						IF aStatCommandQueue[nStatCommandIndex].nSubIndex = 0 THEN
							  nStatOffset := 8;
						END_IF;
							nStatBitLength := 8;
							nTempDeviceDataInteger := UINT_TO_DWORD(stDeviceData.stData.stNetwork.nRoleInNetwork);
							JMP SetInteger;
						END_IF;
					// stNetwork - nDeviceNoMasterHighestNo [UINT] [READ_WRITE]
					IF (aStatCommandQueue[nStatCommandIndex].nSubIndex = 0 AND nStatIndex = 1) OR (aStatCommandQueue[nStatCommandIndex].nSubIndex = 2 AND nStatIndex = 0) THEN
						IF aStatCommandQueue[nStatCommandIndex].nSubIndex = 0 THEN
							  nStatOffset := 0;
						END_IF;
							nStatBitLength := 8;
							nTempDeviceDataInteger := UINT_TO_DWORD(stDeviceData.stData.stNetwork.nDeviceNoMasterHighestNo);
							JMP SetInteger;
						END_IF;
					END_IF;
		END_CASE;
		// Start  FB;
		fbReadWriteReq(bExecute := TRUE, bRW:= bRW, nLen := aStatCommandQueue[nStatCommandIndex].nBitLength, aData := aStatIOLRecords);
		// Next step
		nStatState := cSTATE_AWAIT_RESPONSE;
	END_IF;
// Wait for the command answer
	IF nStatState = cSTATE_AWAIT_RESPONSE THEN
		fbReadWriteReq(bExecute := FALSE, aData := aStatIOLRecords);
		IF bStatBusyMem AND NOT fbReadWriteReq.bBusy THEN
			nStatIndex := 0;
			IF fbReadWriteReq.bError THEN
				RETURN;
			END_IF;
			nStatState := cSTATE_PARSE_RESPONSE;
		END_IF;
	END_IF;
// Interpret command answer
	IF nStatState = cSTATE_PARSE_RESPONSE THEN
		IF NOT bStatRWSave THEN
			CASE aStatCommandQueue[nStatCommandIndex].nIndex OF
				// stDirectParametersPage1 [ComplexT] [READ_WRITE]
					0:
						nStatComplex := cCOMPLEX_RECORD_TYPE;
						nStatComplexDataTypeSize := UINT_TO_INT(aStatCommandQueue[nStatCommandIndex].nBitLength);
						nStatOffset := 0;
						// stDirectParametersPage1 - nReserved_1 [UINT] [READ_ONLY]
						IF (aStatCommandQueue[nStatCommandIndex].nSubIndex = 0 AND nStatIndex = 0) OR (aStatCommandQueue[nStatCommandIndex].nSubIndex = 1 AND nStatIndex = 0) THEN
							IF aStatCommandQueue[nStatCommandIndex].nSubIndex = 0 THEN
								nStatOffset := 120;
							END_IF;
							nStatElement := 23;
							nStatBitLength := 8;
							bStatSource := False;
							JMP GetInteger;
						END_IF;
						// stDirectParametersPage1 - nMasterCycleTime [UINT] [READ_ONLY]
						IF (aStatCommandQueue[nStatCommandIndex].nSubIndex = 0 AND nStatIndex = 1) OR (aStatCommandQueue[nStatCommandIndex].nSubIndex = 2 AND nStatIndex = 0) THEN
							IF aStatCommandQueue[nStatCommandIndex].nSubIndex = 0 THEN
								nStatOffset := 112;
							END_IF;
							nStatElement := 24;
							nStatBitLength := 8;
							bStatSource := False;
							JMP GetInteger;
						END_IF;
						// stDirectParametersPage1 - nMinCycleTime [UINT] [READ_ONLY]
						IF (aStatCommandQueue[nStatCommandIndex].nSubIndex = 0 AND nStatIndex = 2) OR (aStatCommandQueue[nStatCommandIndex].nSubIndex = 3 AND nStatIndex = 0) THEN
							IF aStatCommandQueue[nStatCommandIndex].nSubIndex = 0 THEN
								nStatOffset := 104;
							END_IF;
							nStatElement := 25;
							nStatBitLength := 8;
							bStatSource := False;
							JMP GetInteger;
						END_IF;
						// stDirectParametersPage1 - nMSequenceCapability [UINT] [READ_ONLY]
						IF (aStatCommandQueue[nStatCommandIndex].nSubIndex = 0 AND nStatIndex = 3) OR (aStatCommandQueue[nStatCommandIndex].nSubIndex = 4 AND nStatIndex = 0) THEN
							IF aStatCommandQueue[nStatCommandIndex].nSubIndex = 0 THEN
								nStatOffset := 96;
							END_IF;
							nStatElement := 26;
							nStatBitLength := 8;
							bStatSource := False;
							JMP GetInteger;
						END_IF;
						// stDirectParametersPage1 - nIoLinkRevisionId [UINT] [READ_ONLY]
						IF (aStatCommandQueue[nStatCommandIndex].nSubIndex = 0 AND nStatIndex = 4) OR (aStatCommandQueue[nStatCommandIndex].nSubIndex = 5 AND nStatIndex = 0) THEN
							IF aStatCommandQueue[nStatCommandIndex].nSubIndex = 0 THEN
								nStatOffset := 88;
							END_IF;
							nStatElement := 27;
							nStatBitLength := 8;
							bStatSource := False;
							JMP GetInteger;
						END_IF;
						// stDirectParametersPage1 - nProcessDataInputLength [UINT] [READ_ONLY]
						IF (aStatCommandQueue[nStatCommandIndex].nSubIndex = 0 AND nStatIndex = 5) OR (aStatCommandQueue[nStatCommandIndex].nSubIndex = 6 AND nStatIndex = 0) THEN
							IF aStatCommandQueue[nStatCommandIndex].nSubIndex = 0 THEN
								nStatOffset := 80;
							END_IF;
							nStatElement := 28;
							nStatBitLength := 8;
							bStatSource := False;
							JMP GetInteger;
						END_IF;
						// stDirectParametersPage1 - nProcessDataOutputLength [UINT] [READ_ONLY]
						IF (aStatCommandQueue[nStatCommandIndex].nSubIndex = 0 AND nStatIndex = 6) OR (aStatCommandQueue[nStatCommandIndex].nSubIndex = 7 AND nStatIndex = 0) THEN
							IF aStatCommandQueue[nStatCommandIndex].nSubIndex = 0 THEN
								nStatOffset := 72;
							END_IF;
							nStatElement := 29;
							nStatBitLength := 8;
							bStatSource := False;
							JMP GetInteger;
						END_IF;
						// stDirectParametersPage1 - nVendorId1 [UINT] [READ_ONLY]
						IF (aStatCommandQueue[nStatCommandIndex].nSubIndex = 0 AND nStatIndex = 7) OR (aStatCommandQueue[nStatCommandIndex].nSubIndex = 8 AND nStatIndex = 0) THEN
							IF aStatCommandQueue[nStatCommandIndex].nSubIndex = 0 THEN
								nStatOffset := 64;
							END_IF;
							nStatElement := 30;
							nStatBitLength := 8;
							bStatSource := False;
							JMP GetInteger;
						END_IF;
						// stDirectParametersPage1 - nVendorId2 [UINT] [READ_ONLY]
						IF (aStatCommandQueue[nStatCommandIndex].nSubIndex = 0 AND nStatIndex = 8) OR (aStatCommandQueue[nStatCommandIndex].nSubIndex = 9 AND nStatIndex = 0) THEN
							IF aStatCommandQueue[nStatCommandIndex].nSubIndex = 0 THEN
								nStatOffset := 56;
							END_IF;
							nStatElement := 31;
							nStatBitLength := 8;
							bStatSource := False;
							JMP GetInteger;
						END_IF;
						// stDirectParametersPage1 - nDeviceId1 [UINT] [READ_ONLY]
						IF (aStatCommandQueue[nStatCommandIndex].nSubIndex = 0 AND nStatIndex = 9) OR (aStatCommandQueue[nStatCommandIndex].nSubIndex = 10 AND nStatIndex = 0) THEN
							IF aStatCommandQueue[nStatCommandIndex].nSubIndex = 0 THEN
								nStatOffset := 48;
							END_IF;
							nStatElement := 32;
							nStatBitLength := 8;
							bStatSource := False;
							JMP GetInteger;
						END_IF;
						// stDirectParametersPage1 - nDeviceId2 [UINT] [READ_ONLY]
						IF (aStatCommandQueue[nStatCommandIndex].nSubIndex = 0 AND nStatIndex = 10) OR (aStatCommandQueue[nStatCommandIndex].nSubIndex = 11 AND nStatIndex = 0) THEN
							IF aStatCommandQueue[nStatCommandIndex].nSubIndex = 0 THEN
								nStatOffset := 40;
							END_IF;
							nStatElement := 33;
							nStatBitLength := 8;
							bStatSource := False;
							JMP GetInteger;
						END_IF;
						// stDirectParametersPage1 - nDeviceId3 [UINT] [READ_ONLY]
						IF (aStatCommandQueue[nStatCommandIndex].nSubIndex = 0 AND nStatIndex = 11) OR (aStatCommandQueue[nStatCommandIndex].nSubIndex = 12 AND nStatIndex = 0) THEN
							IF aStatCommandQueue[nStatCommandIndex].nSubIndex = 0 THEN
								nStatOffset := 32;
							END_IF;
							nStatElement := 34;
							nStatBitLength := 8;
							bStatSource := False;
							JMP GetInteger;
						END_IF;
						// stDirectParametersPage1 - nReserved_13 [UINT] [READ_ONLY]
						IF (aStatCommandQueue[nStatCommandIndex].nSubIndex = 0 AND nStatIndex = 12) OR (aStatCommandQueue[nStatCommandIndex].nSubIndex = 13 AND nStatIndex = 0) THEN
							IF aStatCommandQueue[nStatCommandIndex].nSubIndex = 0 THEN
								nStatOffset := 24;
							END_IF;
							nStatElement := 35;
							nStatBitLength := 8;
							bStatSource := False;
							JMP GetInteger;
						END_IF;
						// stDirectParametersPage1 - nReserved_14 [UINT] [READ_ONLY]
						IF (aStatCommandQueue[nStatCommandIndex].nSubIndex = 0 AND nStatIndex = 13) OR (aStatCommandQueue[nStatCommandIndex].nSubIndex = 14 AND nStatIndex = 0) THEN
							IF aStatCommandQueue[nStatCommandIndex].nSubIndex = 0 THEN
								nStatOffset := 16;
							END_IF;
							nStatElement := 36;
							nStatBitLength := 8;
							bStatSource := False;
							JMP GetInteger;
						END_IF;
						// stDirectParametersPage1 - nReserved_15 [UINT] [READ_ONLY]
						IF (aStatCommandQueue[nStatCommandIndex].nSubIndex = 0 AND nStatIndex = 14) OR (aStatCommandQueue[nStatCommandIndex].nSubIndex = 15 AND nStatIndex = 0) THEN
							IF aStatCommandQueue[nStatCommandIndex].nSubIndex = 0 THEN
								nStatOffset := 8;
							END_IF;
							nStatElement := 37;
							nStatBitLength := 8;
							bStatSource := False;
							JMP GetInteger;
						END_IF;
				// stDirectParametersPage2 [ComplexT] [READ_WRITE]
					1:
						nStatComplex := cCOMPLEX_RECORD_TYPE;
						nStatComplexDataTypeSize := UINT_TO_INT(aStatCommandQueue[nStatCommandIndex].nBitLength);
						nStatOffset := 0;
						// stDirectParametersPage2 - nDeviceSpecificParameter1 [UINT] [READ_WRITE]
						IF (aStatCommandQueue[nStatCommandIndex].nSubIndex = 0 AND nStatIndex = 0) OR (aStatCommandQueue[nStatCommandIndex].nSubIndex = 1 AND nStatIndex = 0) THEN
							IF aStatCommandQueue[nStatCommandIndex].nSubIndex = 0 THEN
								nStatOffset := 120;
							END_IF;
							nStatElement := 39;
							nStatBitLength := 8;
							bStatSource := False;
							JMP GetInteger;
						END_IF;
						// stDirectParametersPage2 - nDeviceSpecificParameter2 [UINT] [READ_WRITE]
						IF (aStatCommandQueue[nStatCommandIndex].nSubIndex = 0 AND nStatIndex = 1) OR (aStatCommandQueue[nStatCommandIndex].nSubIndex = 2 AND nStatIndex = 0) THEN
							IF aStatCommandQueue[nStatCommandIndex].nSubIndex = 0 THEN
								nStatOffset := 112;
							END_IF;
							nStatElement := 40;
							nStatBitLength := 8;
							bStatSource := False;
							JMP GetInteger;
						END_IF;
						// stDirectParametersPage2 - nDeviceSpecificParameter3 [UINT] [READ_WRITE]
						IF (aStatCommandQueue[nStatCommandIndex].nSubIndex = 0 AND nStatIndex = 2) OR (aStatCommandQueue[nStatCommandIndex].nSubIndex = 3 AND nStatIndex = 0) THEN
							IF aStatCommandQueue[nStatCommandIndex].nSubIndex = 0 THEN
								nStatOffset := 104;
							END_IF;
							nStatElement := 41;
							nStatBitLength := 8;
							bStatSource := False;
							JMP GetInteger;
						END_IF;
						// stDirectParametersPage2 - nDeviceSpecificParameter4 [UINT] [READ_WRITE]
						IF (aStatCommandQueue[nStatCommandIndex].nSubIndex = 0 AND nStatIndex = 3) OR (aStatCommandQueue[nStatCommandIndex].nSubIndex = 4 AND nStatIndex = 0) THEN
							IF aStatCommandQueue[nStatCommandIndex].nSubIndex = 0 THEN
								nStatOffset := 96;
							END_IF;
							nStatElement := 42;
							nStatBitLength := 8;
							bStatSource := False;
							JMP GetInteger;
						END_IF;
						// stDirectParametersPage2 - nDeviceSpecificParameter5 [UINT] [READ_WRITE]
						IF (aStatCommandQueue[nStatCommandIndex].nSubIndex = 0 AND nStatIndex = 4) OR (aStatCommandQueue[nStatCommandIndex].nSubIndex = 5 AND nStatIndex = 0) THEN
							IF aStatCommandQueue[nStatCommandIndex].nSubIndex = 0 THEN
								nStatOffset := 88;
							END_IF;
							nStatElement := 43;
							nStatBitLength := 8;
							bStatSource := False;
							JMP GetInteger;
						END_IF;
						// stDirectParametersPage2 - nDeviceSpecificParameter6 [UINT] [READ_WRITE]
						IF (aStatCommandQueue[nStatCommandIndex].nSubIndex = 0 AND nStatIndex = 5) OR (aStatCommandQueue[nStatCommandIndex].nSubIndex = 6 AND nStatIndex = 0) THEN
							IF aStatCommandQueue[nStatCommandIndex].nSubIndex = 0 THEN
								nStatOffset := 80;
							END_IF;
							nStatElement := 44;
							nStatBitLength := 8;
							bStatSource := False;
							JMP GetInteger;
						END_IF;
						// stDirectParametersPage2 - nDeviceSpecificParameter7 [UINT] [READ_WRITE]
						IF (aStatCommandQueue[nStatCommandIndex].nSubIndex = 0 AND nStatIndex = 6) OR (aStatCommandQueue[nStatCommandIndex].nSubIndex = 7 AND nStatIndex = 0) THEN
							IF aStatCommandQueue[nStatCommandIndex].nSubIndex = 0 THEN
								nStatOffset := 72;
							END_IF;
							nStatElement := 45;
							nStatBitLength := 8;
							bStatSource := False;
							JMP GetInteger;
						END_IF;
						// stDirectParametersPage2 - nDeviceSpecificParameter8 [UINT] [READ_WRITE]
						IF (aStatCommandQueue[nStatCommandIndex].nSubIndex = 0 AND nStatIndex = 7) OR (aStatCommandQueue[nStatCommandIndex].nSubIndex = 8 AND nStatIndex = 0) THEN
							IF aStatCommandQueue[nStatCommandIndex].nSubIndex = 0 THEN
								nStatOffset := 64;
							END_IF;
							nStatElement := 46;
							nStatBitLength := 8;
							bStatSource := False;
							JMP GetInteger;
						END_IF;
						// stDirectParametersPage2 - nDeviceSpecificParameter9 [UINT] [READ_WRITE]
						IF (aStatCommandQueue[nStatCommandIndex].nSubIndex = 0 AND nStatIndex = 8) OR (aStatCommandQueue[nStatCommandIndex].nSubIndex = 9 AND nStatIndex = 0) THEN
							IF aStatCommandQueue[nStatCommandIndex].nSubIndex = 0 THEN
								nStatOffset := 56;
							END_IF;
							nStatElement := 47;
							nStatBitLength := 8;
							bStatSource := False;
							JMP GetInteger;
						END_IF;
						// stDirectParametersPage2 - nDeviceSpecificParameter10 [UINT] [READ_WRITE]
						IF (aStatCommandQueue[nStatCommandIndex].nSubIndex = 0 AND nStatIndex = 9) OR (aStatCommandQueue[nStatCommandIndex].nSubIndex = 10 AND nStatIndex = 0) THEN
							IF aStatCommandQueue[nStatCommandIndex].nSubIndex = 0 THEN
								nStatOffset := 48;
							END_IF;
							nStatElement := 48;
							nStatBitLength := 8;
							bStatSource := False;
							JMP GetInteger;
						END_IF;
						// stDirectParametersPage2 - nDeviceSpecificParameter11 [UINT] [READ_WRITE]
						IF (aStatCommandQueue[nStatCommandIndex].nSubIndex = 0 AND nStatIndex = 10) OR (aStatCommandQueue[nStatCommandIndex].nSubIndex = 11 AND nStatIndex = 0) THEN
							IF aStatCommandQueue[nStatCommandIndex].nSubIndex = 0 THEN
								nStatOffset := 40;
							END_IF;
							nStatElement := 49;
							nStatBitLength := 8;
							bStatSource := False;
							JMP GetInteger;
						END_IF;
						// stDirectParametersPage2 - nDeviceSpecificParameter12 [UINT] [READ_WRITE]
						IF (aStatCommandQueue[nStatCommandIndex].nSubIndex = 0 AND nStatIndex = 11) OR (aStatCommandQueue[nStatCommandIndex].nSubIndex = 12 AND nStatIndex = 0) THEN
							IF aStatCommandQueue[nStatCommandIndex].nSubIndex = 0 THEN
								nStatOffset := 32;
							END_IF;
							nStatElement := 50;
							nStatBitLength := 8;
							bStatSource := False;
							JMP GetInteger;
						END_IF;
						// stDirectParametersPage2 - nDeviceSpecificParameter13 [UINT] [READ_WRITE]
						IF (aStatCommandQueue[nStatCommandIndex].nSubIndex = 0 AND nStatIndex = 12) OR (aStatCommandQueue[nStatCommandIndex].nSubIndex = 13 AND nStatIndex = 0) THEN
							IF aStatCommandQueue[nStatCommandIndex].nSubIndex = 0 THEN
								nStatOffset := 24;
							END_IF;
							nStatElement := 51;
							nStatBitLength := 8;
							bStatSource := False;
							JMP GetInteger;
						END_IF;
						// stDirectParametersPage2 - nDeviceSpecificParameter14 [UINT] [READ_WRITE]
						IF (aStatCommandQueue[nStatCommandIndex].nSubIndex = 0 AND nStatIndex = 13) OR (aStatCommandQueue[nStatCommandIndex].nSubIndex = 14 AND nStatIndex = 0) THEN
							IF aStatCommandQueue[nStatCommandIndex].nSubIndex = 0 THEN
								nStatOffset := 16;
							END_IF;
							nStatElement := 52;
							nStatBitLength := 8;
							bStatSource := False;
							JMP GetInteger;
						END_IF;
						// stDirectParametersPage2 - nDeviceSpecificParameter15 [UINT] [READ_WRITE]
						IF (aStatCommandQueue[nStatCommandIndex].nSubIndex = 0 AND nStatIndex = 14) OR (aStatCommandQueue[nStatCommandIndex].nSubIndex = 15 AND nStatIndex = 0) THEN
							IF aStatCommandQueue[nStatCommandIndex].nSubIndex = 0 THEN
								nStatOffset := 8;
							END_IF;
							nStatElement := 53;
							nStatBitLength := 8;
							bStatSource := False;
							JMP GetInteger;
						END_IF;
						// stDirectParametersPage2 - nDeviceSpecificParameter16 [UINT] [READ_WRITE]
						IF (aStatCommandQueue[nStatCommandIndex].nSubIndex = 0 AND nStatIndex = 15) OR (aStatCommandQueue[nStatCommandIndex].nSubIndex = 16 AND nStatIndex = 0) THEN
							IF aStatCommandQueue[nStatCommandIndex].nSubIndex = 0 THEN
								nStatOffset := 0;
							END_IF;
							nStatElement := 54;
							nStatBitLength := 8;
							bStatSource := False;
							JMP GetInteger;
						END_IF;
				// stDeviceAccessLocks [ComplexT] [READ_WRITE]
					12:
						nStatComplex := cCOMPLEX_RECORD_TYPE;
						nStatComplexDataTypeSize := UINT_TO_INT(aStatCommandQueue[nStatCommandIndex].nBitLength);
						nStatOffset := 0;
						// stDeviceAccessLocks - bParameterWriteAccess [BOOL] [READ_WRITE]
							IF (aStatCommandQueue[nStatCommandIndex].nSubIndex = 0 AND nStatIndex = 0) THEN
								nStatOffset := 0;
							nStatElement := 56;
							JMP GetBoolean;
						END_IF;
						// stDeviceAccessLocks - bDataStorage [BOOL] [READ_WRITE]
							IF (aStatCommandQueue[nStatCommandIndex].nSubIndex = 0 AND nStatIndex = 1) THEN
								nStatOffset := 1;
							nStatElement := 57;
							JMP GetBoolean;
						END_IF;
						// stDeviceAccessLocks - bLocalParameterization [BOOL] [READ_WRITE]
							IF (aStatCommandQueue[nStatCommandIndex].nSubIndex = 0 AND nStatIndex = 2) THEN
								nStatOffset := 2;
							nStatElement := 58;
							JMP GetBoolean;
						END_IF;
						// stDeviceAccessLocks - bLocalUserInterface [BOOL] [READ_WRITE]
